REGION Network 41: Kích hoạt mô phỏng TT3208_Bon2 khi ở chế độ Sim Mode
   RUNG wire#powerrail
      Contact( "HMI_Sim_Mode" )
      Contact( "TT3208_Bon2_Sim_Req" )
      Coil( "TT3208_Bon2_Sim_Active" )
   END_RUNG
   // the same network as SCL:
   "TT3208_Bon2_Sim_Active" := "HMI_Sim_Mode" AND "TT3208_Bon2_Sim_Req";
END_REGION

REGION Network 42: Đọc giá trị mô phỏng TT3208_Bon2 vào hiệu dụng
   RUNG wire#powerrail
      Contact( "TT3208_Bon2_Sim_Active" )
      { S7_GenerateENO := "TRUE" } Move(in := "TT3208_Bon2_HMI", out1 => "TT3208_Bon2_Eff")
   END_RUNG
   // the same network as SCL:
   IF "TT3208_Bon2_Sim_Active" THEN "TT3208_Bon2_Eff" := "TT3208_Bon2_HMI"; END_IF;
END_REGION

REGION Network 43: Đọc giá trị vật lý TT3208_Bon2 vào hiệu dụng
   RUNG wire#powerrail
      I_Contact( "TT3208_Bon2_Sim_Active" )
      { S7_GenerateENO := "TRUE" } Move(in := "TT3208_Bon2", out1 => "TT3208_Bon2_Eff")
   END_RUNG
   // the same network as SCL:
   IF NOT "TT3208_Bon2_Sim_Active" THEN "TT3208_Bon2_Eff" := "TT3208_Bon2"; END_IF;
END_REGION

REGION Network 44: Kiểm tra hợp lệ Setpoint PLC1
   RUNG wire#powerrail
      { S7_Templates := "SrcType := Real" } GT_Contact(in1 := "HMI_SP_PLC1_Nuoc_Bon1", in2 := 0.0)
      { S7_Templates := "SrcType := Real" } GT_Contact(in1 := "HMI_SP_PLC1_Nuoc_Bon2", in2 := 0.0)
      { S7_Templates := "SrcType := Real" } GT_Contact(in1 := "HMI_SP_PLC1_Toc_Do_Bon1", in2 := 0.0)
      { S7_Templates := "SrcType := Real" } GT_Contact(in1 := "HMI_SP_PLC1_Toc_Do_Bon2_Main", in2 := 0.0)
      { S7_Templates := "SrcType := Real" } GT_Contact(in1 := "HMI_SP_PLC1_Nhiet_Do_Bon2", in2 := 0.0)
      { S7_Templates := "SrcType := Time" } GT_Contact(in1 := "HMI_SP_Time_Khuay_Bon1", in2 := T#0s)
      { S7_Templates := "SrcType := Time" } GT_Contact(in1 := "HMI_SP_Time_Fwd", in2 := T#0s)
      { S7_Templates := "SrcType := Time" } GT_Contact(in1 := "HMI_SP_Time_Rev", in2 := T#0s)
      { S7_Templates := "SrcType := Time" } GT_Contact(in1 := "HMI_SP_Time_Sterilize", in2 := T#0s)
      Coil( "PLC1_SP_Valid" )
   END_RUNG
   // the same network as SCL:
   "PLC1_SP_Valid" := ("HMI_SP_PLC1_Nuoc_Bon1" > 0.0) AND ("HMI_SP_PLC1_Nuoc_Bon2" > 0.0) AND ("HMI_SP_PLC1_Toc_Do_Bon1" > 0.0) AND ("HMI_SP_PLC1_Toc_Do_Bon2_Main" > 0.0) AND ("HMI_SP_PLC1_Nhiet_Do_Bon2" > 0.0) AND ("HMI_SP_Time_Khuay_Bon1" > T#0s) AND ("HMI_SP_Time_Fwd" > T#0s) AND ("HMI_SP_Time_Rev" > T#0s) AND ("HMI_SP_Time_Sterilize" > T#0s);
END_REGION

REGION Network 45: Nhận cạnh lên nút nhấn Start PLC1
   RUNG wire#powerrail
      Contact( "Nut_Khoi_Dong_Eff" )
      P_Trig( "PLC1_Start_Edge_Old" )
      Coil( "PLC1_Start_Edge_Edge" )
   END_RUNG
   // the same network as SCL:
   #_w1 := "Nut_Khoi_Dong_Eff" AND NOT "PLC1_Start_Edge_Old";   // rising edge
   "PLC1_Start_Edge_Old" := "Nut_Khoi_Dong_Eff";
   "PLC1_Start_Edge_Edge" := #_w1;
END_REGION

REGION Network 46: Khởi động chu trình PLC1 - Set Auto Enable
   RUNG wire#powerrail
      { S7_Templates := "SrcType := Int" } EQ_Contact(in1 := "PLC1_State", in2 := 0)
      Contact( "PLC1_Start_Edge_Edge" )
      I_Contact( "PLC1_Loi_Tong" )
      Contact( "PLC1_SP_Valid" )
      S_Coil( "PLC1_Auto_Enable" )
   END_RUNG
   // the same network as SCL:
   IF ("PLC1_State" = 0) AND "PLC1_Start_Edge_Edge" AND NOT "PLC1_Loi_Tong" AND "PLC1_SP_Valid" THEN
       "PLC1_Auto_Enable" := TRUE;
   END_IF;
END_REGION

REGION Network 47: Khởi động chu trình PLC1 - Chuyển sang State 10
   RUNG wire#powerrail
      { S7_Templates := "SrcType := Int" } EQ_Contact(in1 := "PLC1_State", in2 := 0)
      Contact( "PLC1_Start_Edge_Edge" )
      I_Contact( "PLC1_Loi_Tong" )
      Contact( "PLC1_SP_Valid" )
      { S7_GenerateENO := "TRUE" } Move(in := 10, out1 => "PLC1_State")
   END_RUNG
   // the same network as SCL:
   IF ("PLC1_State" = 0) AND "PLC1_Start_Edge_Edge" AND NOT "PLC1_Loi_Tong" AND "PLC1_SP_Valid" THEN
       "PLC1_State" := 10;
   END_IF;
END_REGION

REGION Network 48: Báo lỗi setpoint PLC1 khi bấm Start
   RUNG wire#powerrail
      Contact( "PLC1_Start_Edge_Edge" )
      I_Contact( "PLC1_Loi_Tong" )
      I_Contact( "PLC1_SP_Valid" )
      S_Coil( "PLC1_Loi_Setpoint" )
   END_RUNG
   // the same network as SCL:
   IF "PLC1_Start_Edge_Edge" AND NOT "PLC1_Loi_Tong" AND NOT "PLC1_SP_Valid" THEN
       "PLC1_Loi_Setpoint" := TRUE;
   END_IF;
END_REGION

REGION Network 49: Stop PLC1 từ nút vật lý hoặc HMI
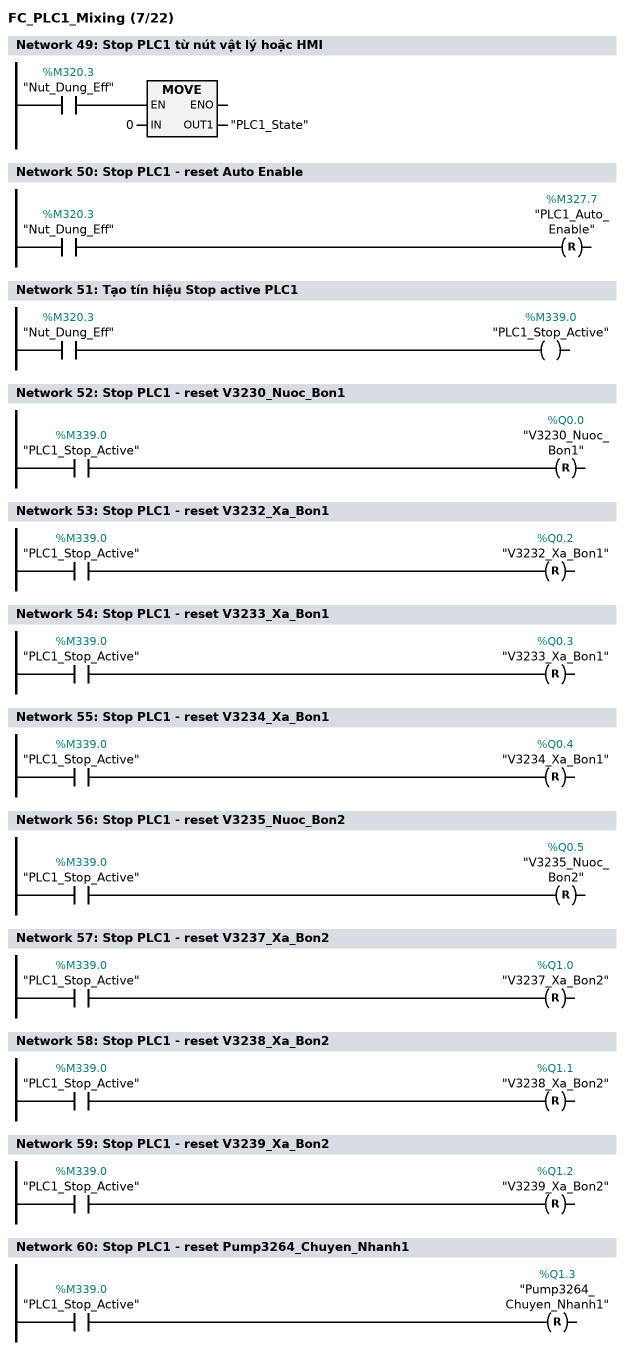
   RUNG wire#powerrail
      Contact( "Nut_Dung_Eff" )
      { S7_GenerateENO := "TRUE" } Move(in := 0, out1 => "PLC1_State")
   END_RUNG
   // the same network as SCL:
   IF "Nut_Dung_Eff" THEN "PLC1_State" := 0; END_IF;
END_REGION

REGION Network 50: Stop PLC1 - reset Auto Enable
   RUNG wire#powerrail
      Contact( "Nut_Dung_Eff" )
      R_Coil( "PLC1_Auto_Enable" )
   END_RUNG
   // the same network as SCL:
   IF "Nut_Dung_Eff" THEN "PLC1_Auto_Enable" := FALSE; END_IF;
END_REGION

REGION Network 51: Tạo tín hiệu Stop active PLC1
   RUNG wire#powerrail
      Contact( "Nut_Dung_Eff" )
      Coil( "PLC1_Stop_Active" )
   END_RUNG
   // the same network as SCL:
   "PLC1_Stop_Active" := "Nut_Dung_Eff";
END_REGION

REGION Network 52: Stop PLC1 - reset V3230_Nuoc_Bon1
   RUNG wire#powerrail
      Contact( "PLC1_Stop_Active" )
      R_Coil( "V3230_Nuoc_Bon1" )
   END_RUNG
   // the same network as SCL:
   IF "PLC1_Stop_Active" THEN "V3230_Nuoc_Bon1" := FALSE; END_IF;
END_REGION

REGION Network 53: Stop PLC1 - reset V3232_Xa_Bon1
   RUNG wire#powerrail
      Contact( "PLC1_Stop_Active" )
      R_Coil( "V3232_Xa_Bon1" )
   END_RUNG
   // the same network as SCL:
   IF "PLC1_Stop_Active" THEN "V3232_Xa_Bon1" := FALSE; END_IF;
END_REGION

REGION Network 54: Stop PLC1 - reset V3233_Xa_Bon1
   RUNG wire#powerrail
      Contact( "PLC1_Stop_Active" )
      R_Coil( "V3233_Xa_Bon1" )
   END_RUNG
   // the same network as SCL:
   IF "PLC1_Stop_Active" THEN "V3233_Xa_Bon1" := FALSE; END_IF;
END_REGION

REGION Network 55: Stop PLC1 - reset V3234_Xa_Bon1
   RUNG wire#powerrail
      Contact( "PLC1_Stop_Active" )
      R_Coil( "V3234_Xa_Bon1" )
   END_RUNG
   // the same network as SCL:
   IF "PLC1_Stop_Active" THEN "V3234_Xa_Bon1" := FALSE; END_IF;
END_REGION

REGION Network 56: Stop PLC1 - reset V3235_Nuoc_Bon2
   RUNG wire#powerrail
      Contact( "PLC1_Stop_Active" )
      R_Coil( "V3235_Nuoc_Bon2" )
   END_RUNG
   // the same network as SCL:
   IF "PLC1_Stop_Active" THEN "V3235_Nuoc_Bon2" := FALSE; END_IF;
END_REGION

REGION Network 57: Stop PLC1 - reset V3237_Xa_Bon2
   RUNG wire#powerrail
      Contact( "PLC1_Stop_Active" )
      R_Coil( "V3237_Xa_Bon2" )
   END_RUNG
   // the same network as SCL:
   IF "PLC1_Stop_Active" THEN "V3237_Xa_Bon2" := FALSE; END_IF;
END_REGION

REGION Network 58: Stop PLC1 - reset V3238_Xa_Bon2
   RUNG wire#powerrail
      Contact( "PLC1_Stop_Active" )
      R_Coil( "V3238_Xa_Bon2" )
   END_RUNG
   // the same network as SCL:
   IF "PLC1_Stop_Active" THEN "V3238_Xa_Bon2" := FALSE; END_IF;
END_REGION

REGION Network 59: Stop PLC1 - reset V3239_Xa_Bon2
   RUNG wire#powerrail
      Contact( "PLC1_Stop_Active" )
      R_Coil( "V3239_Xa_Bon2" )
   END_RUNG
   // the same network as SCL:
   IF "PLC1_Stop_Active" THEN "V3239_Xa_Bon2" := FALSE; END_IF;
END_REGION

REGION Network 60: Stop PLC1 - reset Pump3264_Chuyen_Nhanh1
   RUNG wire#powerrail
      Contact( "PLC1_Stop_Active" )
      R_Coil( "Pump3264_Chuyen_Nhanh1" )
   END_RUNG
   // the same network as SCL:
   IF "PLC1_Stop_Active" THEN "Pump3264_Chuyen_Nhanh1" := FALSE; END_IF;
END_REGION

REGION Network 61: Stop PLC1 - reset PID Enable
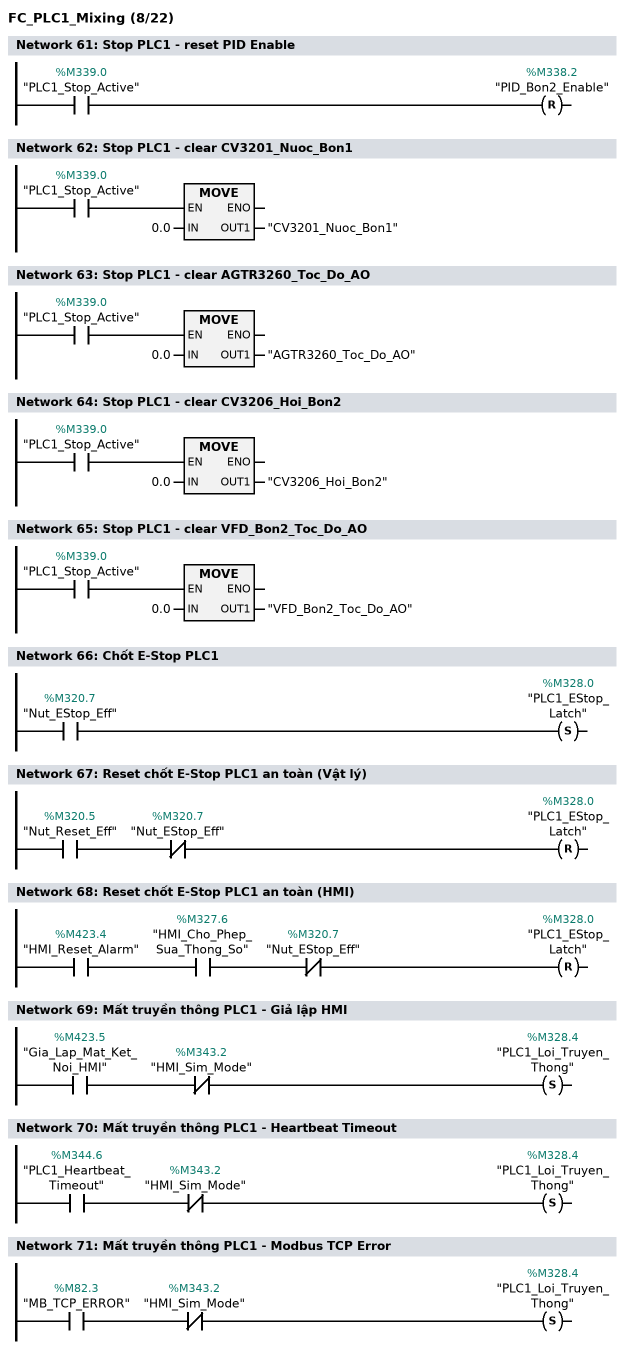
   RUNG wire#powerrail
      Contact( "PLC1_Stop_Active" )
      R_Coil( "PID_Bon2_Enable" )
   END_RUNG
   // the same network as SCL:
   IF "PLC1_Stop_Active" THEN "PID_Bon2_Enable" := FALSE; END_IF;
END_REGION

REGION Network 62: Stop PLC1 - clear CV3201_Nuoc_Bon1
   RUNG wire#powerrail
      Contact( "PLC1_Stop_Active" )
      { S7_GenerateENO := "TRUE" } Move(in := 0.0, out1 => "CV3201_Nuoc_Bon1")
   END_RUNG
   // the same network as SCL:
   IF "PLC1_Stop_Active" THEN "CV3201_Nuoc_Bon1" := 0.0; END_IF;
END_REGION

REGION Network 63: Stop PLC1 - clear AGTR3260_Toc_Do_AO
   RUNG wire#powerrail
      Contact( "PLC1_Stop_Active" )
      { S7_GenerateENO := "TRUE" } Move(in := 0.0, out1 => "AGTR3260_Toc_Do_AO")
   END_RUNG
   // the same network as SCL:
   IF "PLC1_Stop_Active" THEN "AGTR3260_Toc_Do_AO" := 0.0; END_IF;
END_REGION

REGION Network 64: Stop PLC1 - clear CV3206_Hoi_Bon2
   RUNG wire#powerrail
      Contact( "PLC1_Stop_Active" )
      { S7_GenerateENO := "TRUE" } Move(in := 0.0, out1 => "CV3206_Hoi_Bon2")
   END_RUNG
   // the same network as SCL:
   IF "PLC1_Stop_Active" THEN "CV3206_Hoi_Bon2" := 0.0; END_IF;
END_REGION

REGION Network 65: Stop PLC1 - clear VFD_Bon2_Toc_Do_AO
   RUNG wire#powerrail
      Contact( "PLC1_Stop_Active" )
      { S7_GenerateENO := "TRUE" } Move(in := 0.0, out1 => "VFD_Bon2_Toc_Do_AO")
   END_RUNG
   // the same network as SCL:
   IF "PLC1_Stop_Active" THEN "VFD_Bon2_Toc_Do_AO" := 0.0; END_IF;
END_REGION

REGION Network 66: Chốt E-Stop PLC1
   RUNG wire#powerrail
      Contact( "Nut_EStop_Eff" )
      S_Coil( "PLC1_EStop_Latch" )
   END_RUNG
   // the same network as SCL:
   IF "Nut_EStop_Eff" THEN "PLC1_EStop_Latch" := TRUE; END_IF;
END_REGION

REGION Network 67: Reset chốt E-Stop PLC1 an toàn (Vật lý)
   RUNG wire#powerrail
      Contact( "Nut_Reset_Eff" )
      I_Contact( "Nut_EStop_Eff" )
      R_Coil( "PLC1_EStop_Latch" )
   END_RUNG
   // the same network as SCL:
   IF "Nut_Reset_Eff" AND NOT "Nut_EStop_Eff" THEN "PLC1_EStop_Latch" := FALSE; END_IF;
END_REGION

REGION Network 68: Reset chốt E-Stop PLC1 an toàn (HMI)
   RUNG wire#powerrail
      Contact( "HMI_Reset_Alarm" )
      Contact( "HMI_Cho_Phep_Sua_Thong_So" )
      I_Contact( "Nut_EStop_Eff" )
      R_Coil( "PLC1_EStop_Latch" )
   END_RUNG
   // the same network as SCL:
   IF "HMI_Reset_Alarm" AND "HMI_Cho_Phep_Sua_Thong_So" AND NOT "Nut_EStop_Eff" THEN
       "PLC1_EStop_Latch" := FALSE;
   END_IF;
END_REGION

REGION Network 69: Mất truyền thông PLC1 - Giả lập HMI
   RUNG wire#powerrail
      Contact( "Gia_Lap_Mat_Ket_Noi_HMI" )
      I_Contact( "HMI_Sim_Mode" )
      S_Coil( "PLC1_Loi_Truyen_Thong" )
   END_RUNG
   // the same network as SCL:
   IF "Gia_Lap_Mat_Ket_Noi_HMI" AND NOT "HMI_Sim_Mode" THEN "PLC1_Loi_Truyen_Thong" := TRUE; END_IF;
END_REGION

REGION Network 70: Mất truyền thông PLC1 - Heartbeat Timeout
   RUNG wire#powerrail
      Contact( "PLC1_Heartbeat_Timeout" )
      I_Contact( "HMI_Sim_Mode" )
      S_Coil( "PLC1_Loi_Truyen_Thong" )
   END_RUNG
   // the same network as SCL:
   IF "PLC1_Heartbeat_Timeout" AND NOT "HMI_Sim_Mode" THEN "PLC1_Loi_Truyen_Thong" := TRUE; END_IF;
END_REGION

REGION Network 71: Mất truyền thông PLC1 - Modbus TCP Error
   RUNG wire#powerrail
      Contact( "MB_TCP_ERROR" )
      I_Contact( "HMI_Sim_Mode" )
      S_Coil( "PLC1_Loi_Truyen_Thong" )
   END_RUNG
   // the same network as SCL:
   IF "MB_TCP_ERROR" AND NOT "HMI_Sim_Mode" THEN "PLC1_Loi_Truyen_Thong" := TRUE; END_IF;
END_REGION

REGION Network 72: Dry Run bơm Nhánh 1
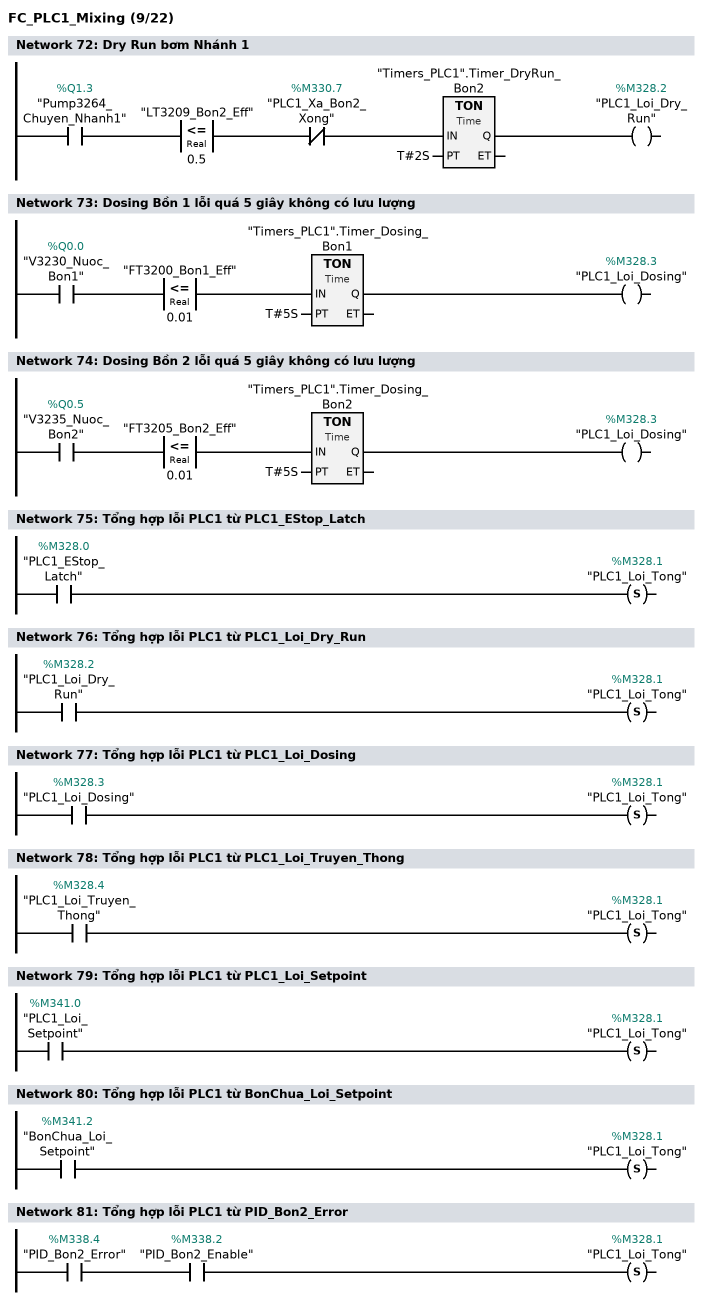
   RUNG wire#powerrail
      Contact( "Pump3264_Chuyen_Nhanh1" )
      { S7_Templates := "SrcType := Real" } LE_Contact(in1 := "LT3209_Bon2_Eff", in2 := 0.5)
      I_Contact( "PLC1_Xa_Bon2_Xong" )
      { S7_Templates := "time_type := Time" } "Timers_PLC1".Timer_DryRun_Bon2.TON(pt := T#2S, et =>)
      Coil( "PLC1_Loi_Dry_Run" )
   END_RUNG
   // the same network as SCL:
   "Timers_PLC1".Timer_DryRun_Bon2.TON(IN := "Pump3264_Chuyen_Nhanh1" AND ("LT3209_Bon2_Eff" <= 0.5) AND NOT "PLC1_Xa_Bon2_Xong",
                           PT := T#2S);
   "PLC1_Loi_Dry_Run" := "Timers_PLC1".Timer_DryRun_Bon2.Q;
END_REGION

REGION Network 73: Dosing Bồn 1 lỗi quá 5 giây không có lưu lượng
   RUNG wire#powerrail
      Contact( "V3230_Nuoc_Bon1" )
      { S7_Templates := "SrcType := Real" } LE_Contact(in1 := "FT3200_Bon1_Eff", in2 := 0.01)
      { S7_Templates := "time_type := Time" } "Timers_PLC1".Timer_Dosing_Bon1.TON(pt := T#5S, et =>)
      Coil( "PLC1_Loi_Dosing" )
   END_RUNG
   // the same network as SCL:
   "Timers_PLC1".Timer_Dosing_Bon1.TON(IN := "V3230_Nuoc_Bon1" AND ("FT3200_Bon1_Eff" <= 0.01), PT := T#5S);
   "PLC1_Loi_Dosing" := "Timers_PLC1".Timer_Dosing_Bon1.Q;
END_REGION

REGION Network 74: Dosing Bồn 2 lỗi quá 5 giây không có lưu lượng
   RUNG wire#powerrail
      Contact( "V3235_Nuoc_Bon2" )
      { S7_Templates := "SrcType := Real" } LE_Contact(in1 := "FT3205_Bon2_Eff", in2 := 0.01)
      { S7_Templates := "time_type := Time" } "Timers_PLC1".Timer_Dosing_Bon2.TON(pt := T#5S, et =>)
      Coil( "PLC1_Loi_Dosing" )
   END_RUNG
   // the same network as SCL:
   "Timers_PLC1".Timer_Dosing_Bon2.TON(IN := "V3235_Nuoc_Bon2" AND ("FT3205_Bon2_Eff" <= 0.01), PT := T#5S);
   "PLC1_Loi_Dosing" := "Timers_PLC1".Timer_Dosing_Bon2.Q;
END_REGION

REGION Network 75: Tổng hợp lỗi PLC1 từ PLC1_EStop_Latch
   RUNG wire#powerrail
      Contact( "PLC1_EStop_Latch" )
      S_Coil( "PLC1_Loi_Tong" )
   END_RUNG
   // the same network as SCL:
   IF "PLC1_EStop_Latch" THEN "PLC1_Loi_Tong" := TRUE; END_IF;
END_REGION

REGION Network 76: Tổng hợp lỗi PLC1 từ PLC1_Loi_Dry_Run
   RUNG wire#powerrail
      Contact( "PLC1_Loi_Dry_Run" )
      S_Coil( "PLC1_Loi_Tong" )
   END_RUNG
   // the same network as SCL:
   IF "PLC1_Loi_Dry_Run" THEN "PLC1_Loi_Tong" := TRUE; END_IF;
END_REGION

REGION Network 77: Tổng hợp lỗi PLC1 từ PLC1_Loi_Dosing
   RUNG wire#powerrail
      Contact( "PLC1_Loi_Dosing" )
      S_Coil( "PLC1_Loi_Tong" )
   END_RUNG
   // the same network as SCL:
   IF "PLC1_Loi_Dosing" THEN "PLC1_Loi_Tong" := TRUE; END_IF;
END_REGION

REGION Network 78: Tổng hợp lỗi PLC1 từ PLC1_Loi_Truyen_Thong
   RUNG wire#powerrail
      Contact( "PLC1_Loi_Truyen_Thong" )
      S_Coil( "PLC1_Loi_Tong" )
   END_RUNG
   // the same network as SCL:
   IF "PLC1_Loi_Truyen_Thong" THEN "PLC1_Loi_Tong" := TRUE; END_IF;
END_REGION

REGION Network 79: Tổng hợp lỗi PLC1 từ PLC1_Loi_Setpoint
   RUNG wire#powerrail
      Contact( "PLC1_Loi_Setpoint" )
      S_Coil( "PLC1_Loi_Tong" )
   END_RUNG
   // the same network as SCL:
   IF "PLC1_Loi_Setpoint" THEN "PLC1_Loi_Tong" := TRUE; END_IF;
END_REGION

REGION Network 80: Tổng hợp lỗi PLC1 từ BonChua_Loi_Setpoint
   RUNG wire#powerrail
      Contact( "BonChua_Loi_Setpoint" )
      S_Coil( "PLC1_Loi_Tong" )
   END_RUNG
   // the same network as SCL:
   IF "BonChua_Loi_Setpoint" THEN "PLC1_Loi_Tong" := TRUE; END_IF;
END_REGION

REGION Network 81: Tổng hợp lỗi PLC1 từ PID_Bon2_Error
   RUNG wire#powerrail
      Contact( "PID_Bon2_Error" )
      Contact( "PID_Bon2_Enable" )
      S_Coil( "PLC1_Loi_Tong" )
   END_RUNG
   // the same network as SCL:
   IF "PID_Bon2_Error" AND "PID_Bon2_Enable" THEN "PLC1_Loi_Tong" := TRUE; END_IF;
END_REGION

REGION Network 82: Tổng hợp lỗi PLC1 từ VFD_Bon2_MB_Error
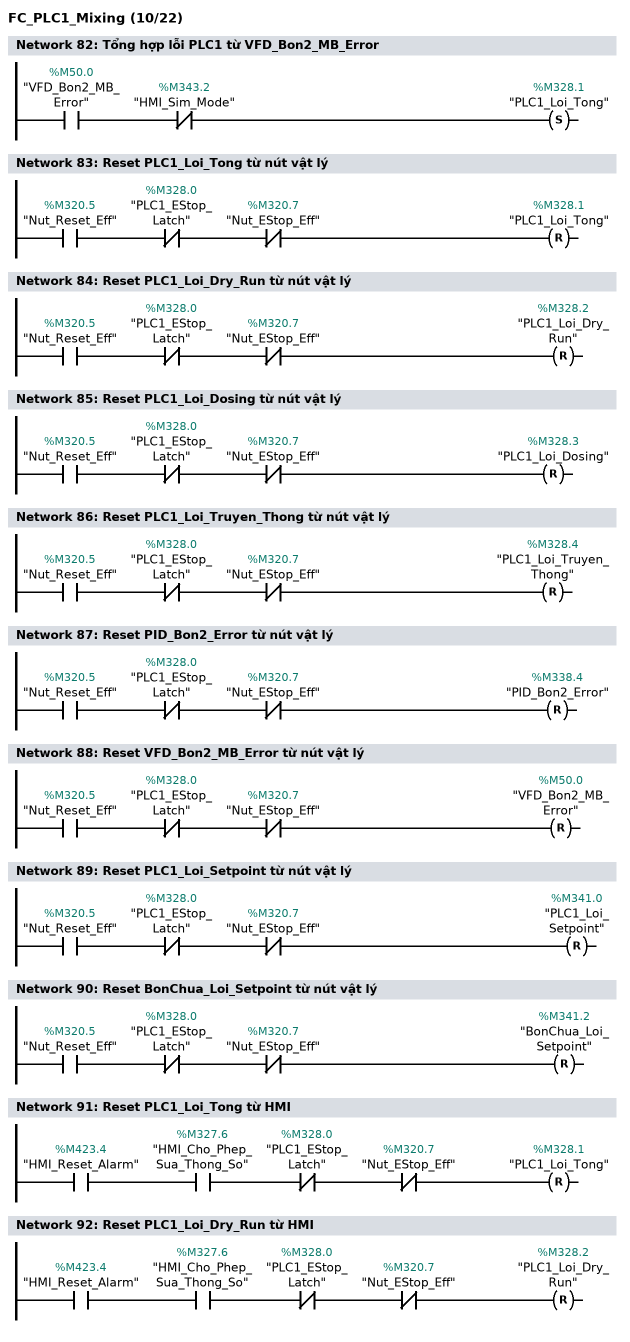
   RUNG wire#powerrail
      Contact( "VFD_Bon2_MB_Error" )
      I_Contact( "HMI_Sim_Mode" )
      S_Coil( "PLC1_Loi_Tong" )
   END_RUNG
   // the same network as SCL:
   IF "VFD_Bon2_MB_Error" AND NOT "HMI_Sim_Mode" THEN "PLC1_Loi_Tong" := TRUE; END_IF;
END_REGION

REGION Network 83: Reset PLC1_Loi_Tong từ nút vật lý
   RUNG wire#powerrail
      Contact( "Nut_Reset_Eff" )
      I_Contact( "PLC1_EStop_Latch" )
      I_Contact( "Nut_EStop_Eff" )
      R_Coil( "PLC1_Loi_Tong" )
   END_RUNG
   // the same network as SCL:
   IF "Nut_Reset_Eff" AND NOT "PLC1_EStop_Latch" AND NOT "Nut_EStop_Eff" THEN
       "PLC1_Loi_Tong" := FALSE;
   END_IF;
END_REGION

REGION Network 84: Reset PLC1_Loi_Dry_Run từ nút vật lý
   RUNG wire#powerrail
      Contact( "Nut_Reset_Eff" )
      I_Contact( "PLC1_EStop_Latch" )
      I_Contact( "Nut_EStop_Eff" )
      R_Coil( "PLC1_Loi_Dry_Run" )
   END_RUNG
   // the same network as SCL:
   IF "Nut_Reset_Eff" AND NOT "PLC1_EStop_Latch" AND NOT "Nut_EStop_Eff" THEN
       "PLC1_Loi_Dry_Run" := FALSE;
   END_IF;
END_REGION

REGION Network 85: Reset PLC1_Loi_Dosing từ nút vật lý
   RUNG wire#powerrail
      Contact( "Nut_Reset_Eff" )
      I_Contact( "PLC1_EStop_Latch" )
      I_Contact( "Nut_EStop_Eff" )
      R_Coil( "PLC1_Loi_Dosing" )
   END_RUNG
   // the same network as SCL:
   IF "Nut_Reset_Eff" AND NOT "PLC1_EStop_Latch" AND NOT "Nut_EStop_Eff" THEN
       "PLC1_Loi_Dosing" := FALSE;
   END_IF;
END_REGION

REGION Network 86: Reset PLC1_Loi_Truyen_Thong từ nút vật lý
   RUNG wire#powerrail
      Contact( "Nut_Reset_Eff" )
      I_Contact( "PLC1_EStop_Latch" )
      I_Contact( "Nut_EStop_Eff" )
      R_Coil( "PLC1_Loi_Truyen_Thong" )
   END_RUNG
   // the same network as SCL:
   IF "Nut_Reset_Eff" AND NOT "PLC1_EStop_Latch" AND NOT "Nut_EStop_Eff" THEN
       "PLC1_Loi_Truyen_Thong" := FALSE;
   END_IF;
END_REGION

REGION Network 87: Reset PID_Bon2_Error từ nút vật lý
   RUNG wire#powerrail
      Contact( "Nut_Reset_Eff" )
      I_Contact( "PLC1_EStop_Latch" )
      I_Contact( "Nut_EStop_Eff" )
      R_Coil( "PID_Bon2_Error" )
   END_RUNG
   // the same network as SCL:
   IF "Nut_Reset_Eff" AND NOT "PLC1_EStop_Latch" AND NOT "Nut_EStop_Eff" THEN
       "PID_Bon2_Error" := FALSE;
   END_IF;
END_REGION

REGION Network 88: Reset VFD_Bon2_MB_Error từ nút vật lý
   RUNG wire#powerrail
      Contact( "Nut_Reset_Eff" )
      I_Contact( "PLC1_EStop_Latch" )
      I_Contact( "Nut_EStop_Eff" )
      R_Coil( "VFD_Bon2_MB_Error" )
   END_RUNG
   // the same network as SCL:
   IF "Nut_Reset_Eff" AND NOT "PLC1_EStop_Latch" AND NOT "Nut_EStop_Eff" THEN
       "VFD_Bon2_MB_Error" := FALSE;
   END_IF;
END_REGION

REGION Network 89: Reset PLC1_Loi_Setpoint từ nút vật lý
   RUNG wire#powerrail
      Contact( "Nut_Reset_Eff" )
      I_Contact( "PLC1_EStop_Latch" )
      I_Contact( "Nut_EStop_Eff" )
      R_Coil( "PLC1_Loi_Setpoint" )
   END_RUNG
   // the same network as SCL:
   IF "Nut_Reset_Eff" AND NOT "PLC1_EStop_Latch" AND NOT "Nut_EStop_Eff" THEN
       "PLC1_Loi_Setpoint" := FALSE;
   END_IF;
END_REGION

REGION Network 90: Reset BonChua_Loi_Setpoint từ nút vật lý
   RUNG wire#powerrail
      Contact( "Nut_Reset_Eff" )
      I_Contact( "PLC1_EStop_Latch" )
      I_Contact( "Nut_EStop_Eff" )
      R_Coil( "BonChua_Loi_Setpoint" )
   END_RUNG
   // the same network as SCL:
   IF "Nut_Reset_Eff" AND NOT "PLC1_EStop_Latch" AND NOT "Nut_EStop_Eff" THEN
       "BonChua_Loi_Setpoint" := FALSE;
   END_IF;
END_REGION

REGION Network 91: Reset PLC1_Loi_Tong từ HMI
   RUNG wire#powerrail
      Contact( "HMI_Reset_Alarm" )
      Contact( "HMI_Cho_Phep_Sua_Thong_So" )
      I_Contact( "PLC1_EStop_Latch" )
      I_Contact( "Nut_EStop_Eff" )
      R_Coil( "PLC1_Loi_Tong" )
   END_RUNG
   // the same network as SCL:
   IF "HMI_Reset_Alarm" AND "HMI_Cho_Phep_Sua_Thong_So" AND NOT "PLC1_EStop_Latch" AND NOT "Nut_EStop_Eff" THEN
       "PLC1_Loi_Tong" := FALSE;
   END_IF;
END_REGION

REGION Network 92: Reset PLC1_Loi_Dry_Run từ HMI
   RUNG wire#powerrail
      Contact( "HMI_Reset_Alarm" )
      Contact( "HMI_Cho_Phep_Sua_Thong_So" )
      I_Contact( "PLC1_EStop_Latch" )
      I_Contact( "Nut_EStop_Eff" )
      R_Coil( "PLC1_Loi_Dry_Run" )
   END_RUNG
   // the same network as SCL:
   IF "HMI_Reset_Alarm" AND "HMI_Cho_Phep_Sua_Thong_So" AND NOT "PLC1_EStop_Latch" AND NOT "Nut_EStop_Eff" THEN
       "PLC1_Loi_Dry_Run" := FALSE;
   END_IF;
END_REGION

REGION Network 93: Reset PLC1_Loi_Dosing từ HMI
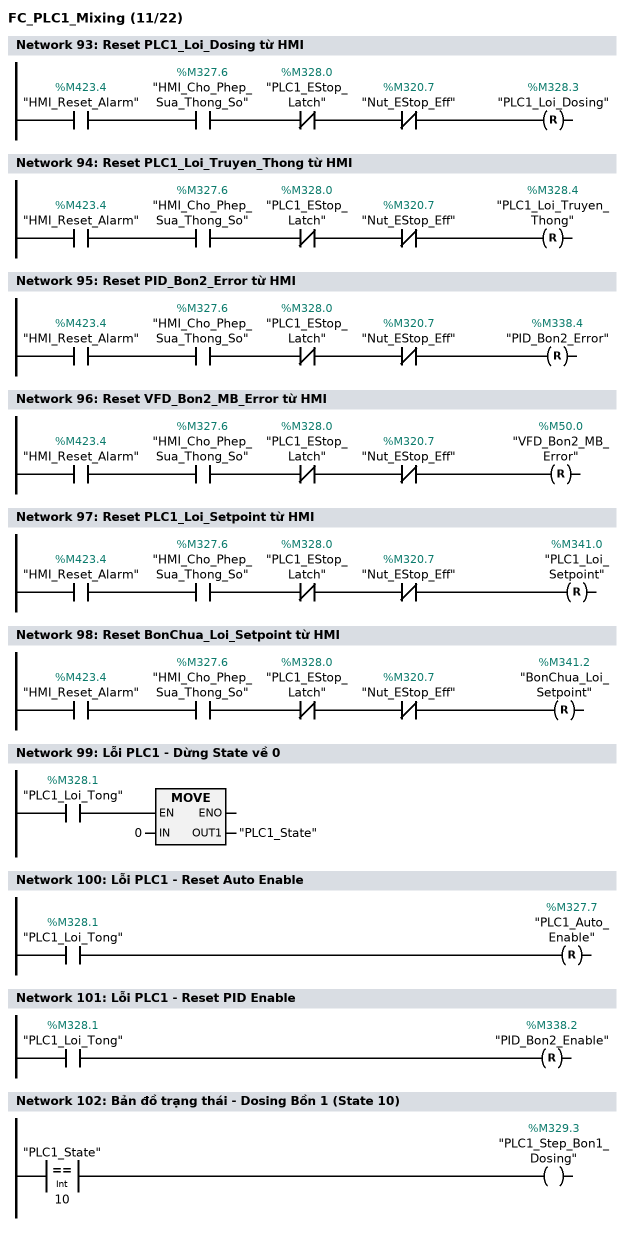
   RUNG wire#powerrail
      Contact( "HMI_Reset_Alarm" )
      Contact( "HMI_Cho_Phep_Sua_Thong_So" )
      I_Contact( "PLC1_EStop_Latch" )
      I_Contact( "Nut_EStop_Eff" )
      R_Coil( "PLC1_Loi_Dosing" )
   END_RUNG
   // the same network as SCL:
   IF "HMI_Reset_Alarm" AND "HMI_Cho_Phep_Sua_Thong_So" AND NOT "PLC1_EStop_Latch" AND NOT "Nut_EStop_Eff" THEN
       "PLC1_Loi_Dosing" := FALSE;
   END_IF;
END_REGION

REGION Network 94: Reset PLC1_Loi_Truyen_Thong từ HMI
   RUNG wire#powerrail
      Contact( "HMI_Reset_Alarm" )
      Contact( "HMI_Cho_Phep_Sua_Thong_So" )
      I_Contact( "PLC1_EStop_Latch" )
      I_Contact( "Nut_EStop_Eff" )
      R_Coil( "PLC1_Loi_Truyen_Thong" )
   END_RUNG
   // the same network as SCL:
   IF "HMI_Reset_Alarm" AND "HMI_Cho_Phep_Sua_Thong_So" AND NOT "PLC1_EStop_Latch" AND NOT "Nut_EStop_Eff" THEN
       "PLC1_Loi_Truyen_Thong" := FALSE;
   END_IF;
END_REGION

REGION Network 95: Reset PID_Bon2_Error từ HMI
   RUNG wire#powerrail
      Contact( "HMI_Reset_Alarm" )
      Contact( "HMI_Cho_Phep_Sua_Thong_So" )
      I_Contact( "PLC1_EStop_Latch" )
      I_Contact( "Nut_EStop_Eff" )
      R_Coil( "PID_Bon2_Error" )
   END_RUNG
   // the same network as SCL:
   IF "HMI_Reset_Alarm" AND "HMI_Cho_Phep_Sua_Thong_So" AND NOT "PLC1_EStop_Latch" AND NOT "Nut_EStop_Eff" THEN
       "PID_Bon2_Error" := FALSE;
   END_IF;
END_REGION

REGION Network 96: Reset VFD_Bon2_MB_Error từ HMI
   RUNG wire#powerrail
      Contact( "HMI_Reset_Alarm" )
      Contact( "HMI_Cho_Phep_Sua_Thong_So" )
      I_Contact( "PLC1_EStop_Latch" )
      I_Contact( "Nut_EStop_Eff" )
      R_Coil( "VFD_Bon2_MB_Error" )
   END_RUNG
   // the same network as SCL:
   IF "HMI_Reset_Alarm" AND "HMI_Cho_Phep_Sua_Thong_So" AND NOT "PLC1_EStop_Latch" AND NOT "Nut_EStop_Eff" THEN
       "VFD_Bon2_MB_Error" := FALSE;
   END_IF;
END_REGION

REGION Network 97: Reset PLC1_Loi_Setpoint từ HMI
   RUNG wire#powerrail
      Contact( "HMI_Reset_Alarm" )
      Contact( "HMI_Cho_Phep_Sua_Thong_So" )
      I_Contact( "PLC1_EStop_Latch" )
      I_Contact( "Nut_EStop_Eff" )
      R_Coil( "PLC1_Loi_Setpoint" )
   END_RUNG
   // the same network as SCL:
   IF "HMI_Reset_Alarm" AND "HMI_Cho_Phep_Sua_Thong_So" AND NOT "PLC1_EStop_Latch" AND NOT "Nut_EStop_Eff" THEN
       "PLC1_Loi_Setpoint" := FALSE;
   END_IF;
END_REGION

REGION Network 98: Reset BonChua_Loi_Setpoint từ HMI
   RUNG wire#powerrail
      Contact( "HMI_Reset_Alarm" )
      Contact( "HMI_Cho_Phep_Sua_Thong_So" )
      I_Contact( "PLC1_EStop_Latch" )
      I_Contact( "Nut_EStop_Eff" )
      R_Coil( "BonChua_Loi_Setpoint" )
   END_RUNG
   // the same network as SCL:
   IF "HMI_Reset_Alarm" AND "HMI_Cho_Phep_Sua_Thong_So" AND NOT "PLC1_EStop_Latch" AND NOT "Nut_EStop_Eff" THEN
       "BonChua_Loi_Setpoint" := FALSE;
   END_IF;
END_REGION

REGION Network 99: Lỗi PLC1 - Dừng State về 0
   RUNG wire#powerrail
      Contact( "PLC1_Loi_Tong" )
      { S7_GenerateENO := "TRUE" } Move(in := 0, out1 => "PLC1_State")
   END_RUNG
   // the same network as SCL:
   IF "PLC1_Loi_Tong" THEN "PLC1_State" := 0; END_IF;
END_REGION

REGION Network 100: Lỗi PLC1 - Reset Auto Enable
   RUNG wire#powerrail
      Contact( "PLC1_Loi_Tong" )
      R_Coil( "PLC1_Auto_Enable" )
   END_RUNG
   // the same network as SCL:
   IF "PLC1_Loi_Tong" THEN "PLC1_Auto_Enable" := FALSE; END_IF;
END_REGION

REGION Network 101: Lỗi PLC1 - Reset PID Enable
   RUNG wire#powerrail
      Contact( "PLC1_Loi_Tong" )
      R_Coil( "PID_Bon2_Enable" )
   END_RUNG
   // the same network as SCL:
   IF "PLC1_Loi_Tong" THEN "PID_Bon2_Enable" := FALSE; END_IF;
END_REGION

REGION Network 102: Bản đồ trạng thái - Dosing Bồn 1 (State 10)
   RUNG wire#powerrail
      { S7_Templates := "SrcType := Int" } EQ_Contact(in1 := "PLC1_State", in2 := 10)
      Coil( "PLC1_Step_Bon1_Dosing" )
   END_RUNG
   // the same network as SCL:
   "PLC1_Step_Bon1_Dosing" := "PLC1_State" = 10;
END_REGION

REGION Network 103: Bản đồ trạng thái - Tip Bồn 1 (State 11)
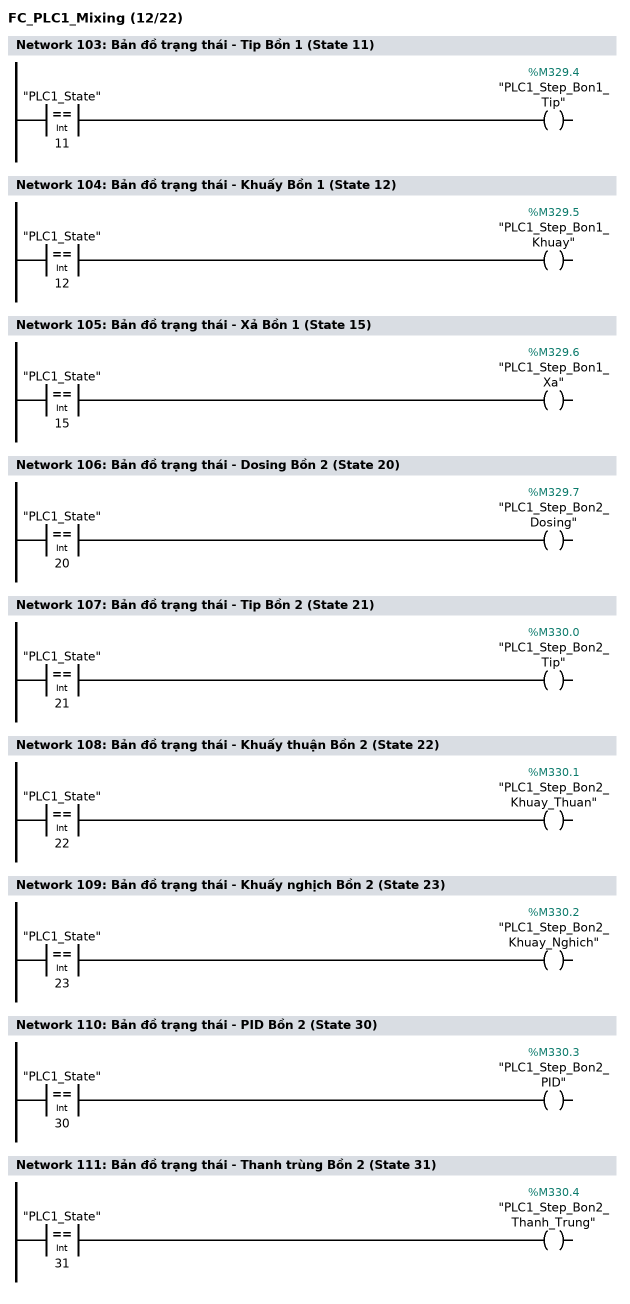
   RUNG wire#powerrail
      { S7_Templates := "SrcType := Int" } EQ_Contact(in1 := "PLC1_State", in2 := 11)
      Coil( "PLC1_Step_Bon1_Tip" )
   END_RUNG
   // the same network as SCL:
   "PLC1_Step_Bon1_Tip" := "PLC1_State" = 11;
END_REGION

REGION Network 104: Bản đồ trạng thái - Khuấy Bồn 1 (State 12)
   RUNG wire#powerrail
      { S7_Templates := "SrcType := Int" } EQ_Contact(in1 := "PLC1_State", in2 := 12)
      Coil( "PLC1_Step_Bon1_Khuay" )
   END_RUNG
   // the same network as SCL:
   "PLC1_Step_Bon1_Khuay" := "PLC1_State" = 12;
END_REGION

REGION Network 105: Bản đồ trạng thái - Xả Bồn 1 (State 15)
   RUNG wire#powerrail
      { S7_Templates := "SrcType := Int" } EQ_Contact(in1 := "PLC1_State", in2 := 15)
      Coil( "PLC1_Step_Bon1_Xa" )
   END_RUNG
   // the same network as SCL:
   "PLC1_Step_Bon1_Xa" := "PLC1_State" = 15;
END_REGION

REGION Network 106: Bản đồ trạng thái - Dosing Bồn 2 (State 20)
   RUNG wire#powerrail
      { S7_Templates := "SrcType := Int" } EQ_Contact(in1 := "PLC1_State", in2 := 20)
      Coil( "PLC1_Step_Bon2_Dosing" )
   END_RUNG
   // the same network as SCL:
   "PLC1_Step_Bon2_Dosing" := "PLC1_State" = 20;
END_REGION

REGION Network 107: Bản đồ trạng thái - Tip Bồn 2 (State 21)
   RUNG wire#powerrail
      { S7_Templates := "SrcType := Int" } EQ_Contact(in1 := "PLC1_State", in2 := 21)
      Coil( "PLC1_Step_Bon2_Tip" )
   END_RUNG
   // the same network as SCL:
   "PLC1_Step_Bon2_Tip" := "PLC1_State" = 21;
END_REGION

REGION Network 108: Bản đồ trạng thái - Khuấy thuận Bồn 2 (State 22)
   RUNG wire#powerrail
      { S7_Templates := "SrcType := Int" } EQ_Contact(in1 := "PLC1_State", in2 := 22)
      Coil( "PLC1_Step_Bon2_Khuay_Thuan" )
   END_RUNG
   // the same network as SCL:
   "PLC1_Step_Bon2_Khuay_Thuan" := "PLC1_State" = 22;
END_REGION

REGION Network 109: Bản đồ trạng thái - Khuấy nghịch Bồn 2 (State 23)
   RUNG wire#powerrail
      { S7_Templates := "SrcType := Int" } EQ_Contact(in1 := "PLC1_State", in2 := 23)
      Coil( "PLC1_Step_Bon2_Khuay_Nghich" )
   END_RUNG
   // the same network as SCL:
   "PLC1_Step_Bon2_Khuay_Nghich" := "PLC1_State" = 23;
END_REGION

REGION Network 110: Bản đồ trạng thái - PID Bồn 2 (State 30)
   RUNG wire#powerrail
      { S7_Templates := "SrcType := Int" } EQ_Contact(in1 := "PLC1_State", in2 := 30)
      Coil( "PLC1_Step_Bon2_PID" )
   END_RUNG
   // the same network as SCL:
   "PLC1_Step_Bon2_PID" := "PLC1_State" = 30;
END_REGION

REGION Network 111: Bản đồ trạng thái - Thanh trùng Bồn 2 (State 31)
   RUNG wire#powerrail
      { S7_Templates := "SrcType := Int" } EQ_Contact(in1 := "PLC1_State", in2 := 31)
      Coil( "PLC1_Step_Bon2_Thanh_Trung" )
   END_RUNG
   // the same network as SCL:
   "PLC1_Step_Bon2_Thanh_Trung" := "PLC1_State" = 31;
END_REGION

REGION Network 112: Bản đồ trạng thái - Nhánh 1 Hoàn thành (State 40)
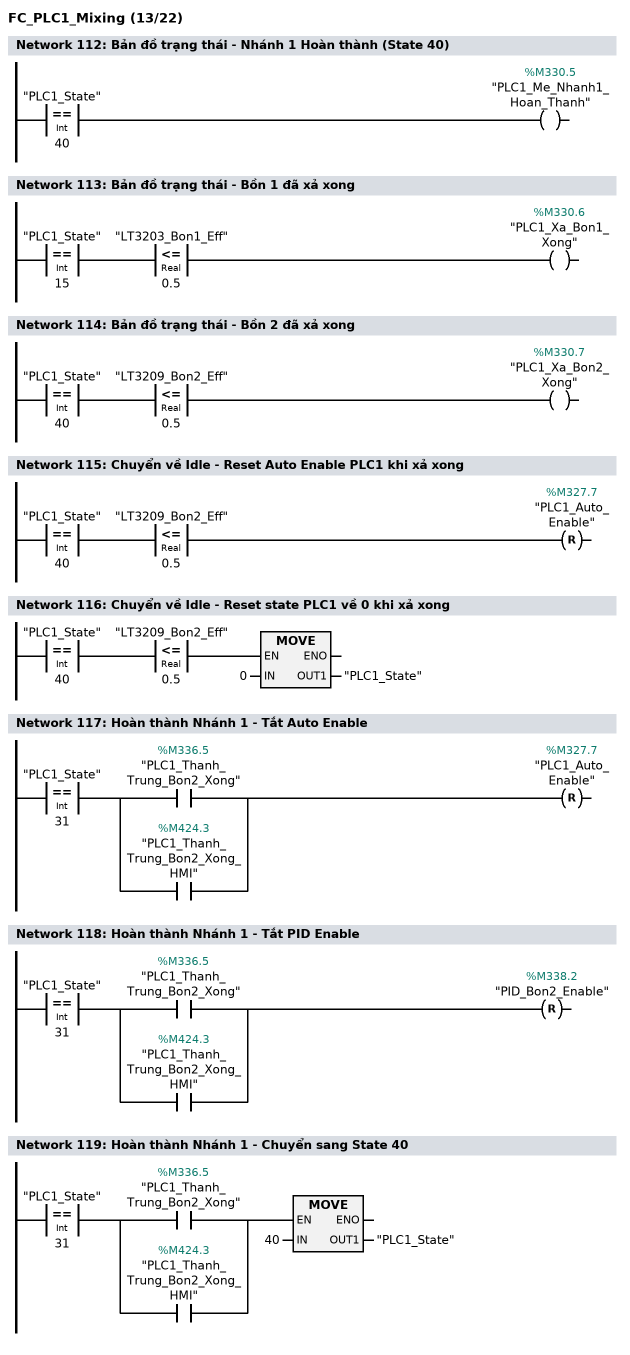
   RUNG wire#powerrail
      { S7_Templates := "SrcType := Int" } EQ_Contact(in1 := "PLC1_State", in2 := 40)
      Coil( "PLC1_Me_Nhanh1_Hoan_Thanh" )
   END_RUNG
   // the same network as SCL:
   "PLC1_Me_Nhanh1_Hoan_Thanh" := "PLC1_State" = 40;
END_REGION

REGION Network 113: Bản đồ trạng thái - Bồn 1 đã xả xong
   RUNG wire#powerrail
      { S7_Templates := "SrcType := Int" } EQ_Contact(in1 := "PLC1_State", in2 := 15)
      { S7_Templates := "SrcType := Real" } LE_Contact(in1 := "LT3203_Bon1_Eff", in2 := 0.5)
      Coil( "PLC1_Xa_Bon1_Xong" )
   END_RUNG
   // the same network as SCL:
   "PLC1_Xa_Bon1_Xong" := ("PLC1_State" = 15) AND ("LT3203_Bon1_Eff" <= 0.5);
END_REGION

REGION Network 114: Bản đồ trạng thái - Bồn 2 đã xả xong
   RUNG wire#powerrail
      { S7_Templates := "SrcType := Int" } EQ_Contact(in1 := "PLC1_State", in2 := 40)
      { S7_Templates := "SrcType := Real" } LE_Contact(in1 := "LT3209_Bon2_Eff", in2 := 0.5)
      Coil( "PLC1_Xa_Bon2_Xong" )
   END_RUNG
   // the same network as SCL:
   "PLC1_Xa_Bon2_Xong" := ("PLC1_State" = 40) AND ("LT3209_Bon2_Eff" <= 0.5);
END_REGION

REGION Network 115: Chuyển về Idle - Reset Auto Enable PLC1 khi xả xong
   RUNG wire#powerrail
      { S7_Templates := "SrcType := Int" } EQ_Contact(in1 := "PLC1_State", in2 := 40)
      { S7_Templates := "SrcType := Real" } LE_Contact(in1 := "LT3209_Bon2_Eff", in2 := 0.5)
      R_Coil( "PLC1_Auto_Enable" )
   END_RUNG
   // the same network as SCL:
   IF ("PLC1_State" = 40) AND ("LT3209_Bon2_Eff" <= 0.5) THEN "PLC1_Auto_Enable" := FALSE; END_IF;
END_REGION

REGION Network 116: Chuyển về Idle - Reset state PLC1 về 0 khi xả xong
   RUNG wire#powerrail
      { S7_Templates := "SrcType := Int" } EQ_Contact(in1 := "PLC1_State", in2 := 40)
      { S7_Templates := "SrcType := Real" } LE_Contact(in1 := "LT3209_Bon2_Eff", in2 := 0.5)
      { S7_GenerateENO := "TRUE" } Move(in := 0, out1 => "PLC1_State")
   END_RUNG
   // the same network as SCL:
   IF ("PLC1_State" = 40) AND ("LT3209_Bon2_Eff" <= 0.5) THEN "PLC1_State" := 0; END_IF;
END_REGION

REGION Network 117: Hoàn thành Nhánh 1 - Tắt Auto Enable
   RUNG wire#powerrail
      { S7_Templates := "SrcType := Int" } EQ_Contact(in1 := "PLC1_State", in2 := 31)
      wire#w1
      Contact( "PLC1_Thanh_Trung_Bon2_Xong" )
      wire#w2
      R_Coil( "PLC1_Auto_Enable" )
   END_RUNG
   RUNG wire#w1
      Contact( "PLC1_Thanh_Trung_Bon2_Xong_HMI" )
   END_RUNG wire#w2
   // the same network as SCL:
   IF ("PLC1_State" = 31) AND ("PLC1_Thanh_Trung_Bon2_Xong" OR "PLC1_Thanh_Trung_Bon2_Xong_HMI") THEN
       "PLC1_Auto_Enable" := FALSE;
   END_IF;
END_REGION

REGION Network 118: Hoàn thành Nhánh 1 - Tắt PID Enable
   RUNG wire#powerrail
      { S7_Templates := "SrcType := Int" } EQ_Contact(in1 := "PLC1_State", in2 := 31)
      wire#w1
      Contact( "PLC1_Thanh_Trung_Bon2_Xong" )
      wire#w2
      R_Coil( "PID_Bon2_Enable" )
   END_RUNG
   RUNG wire#w1
      Contact( "PLC1_Thanh_Trung_Bon2_Xong_HMI" )
   END_RUNG wire#w2
   // the same network as SCL:
   IF ("PLC1_State" = 31) AND ("PLC1_Thanh_Trung_Bon2_Xong" OR "PLC1_Thanh_Trung_Bon2_Xong_HMI") THEN
       "PID_Bon2_Enable" := FALSE;
   END_IF;
END_REGION

REGION Network 119: Hoàn thành Nhánh 1 - Chuyển sang State 40
   RUNG wire#powerrail
      { S7_Templates := "SrcType := Int" } EQ_Contact(in1 := "PLC1_State", in2 := 31)
      wire#w1
      Contact( "PLC1_Thanh_Trung_Bon2_Xong" )
      wire#w2
      { S7_GenerateENO := "TRUE" } Move(in := 40, out1 => "PLC1_State")
   END_RUNG
   RUNG wire#w1
      Contact( "PLC1_Thanh_Trung_Bon2_Xong_HMI" )
   END_RUNG wire#w2
   // the same network as SCL:
   IF ("PLC1_State" = 31) AND ("PLC1_Thanh_Trung_Bon2_Xong" OR "PLC1_Thanh_Trung_Bon2_Xong_HMI") THEN
       "PLC1_State" := 40;
   END_IF;
END_REGION

REGION Network 120: Gia nhiệt Bồn 2 đạt SP - Chuyển sang State 31
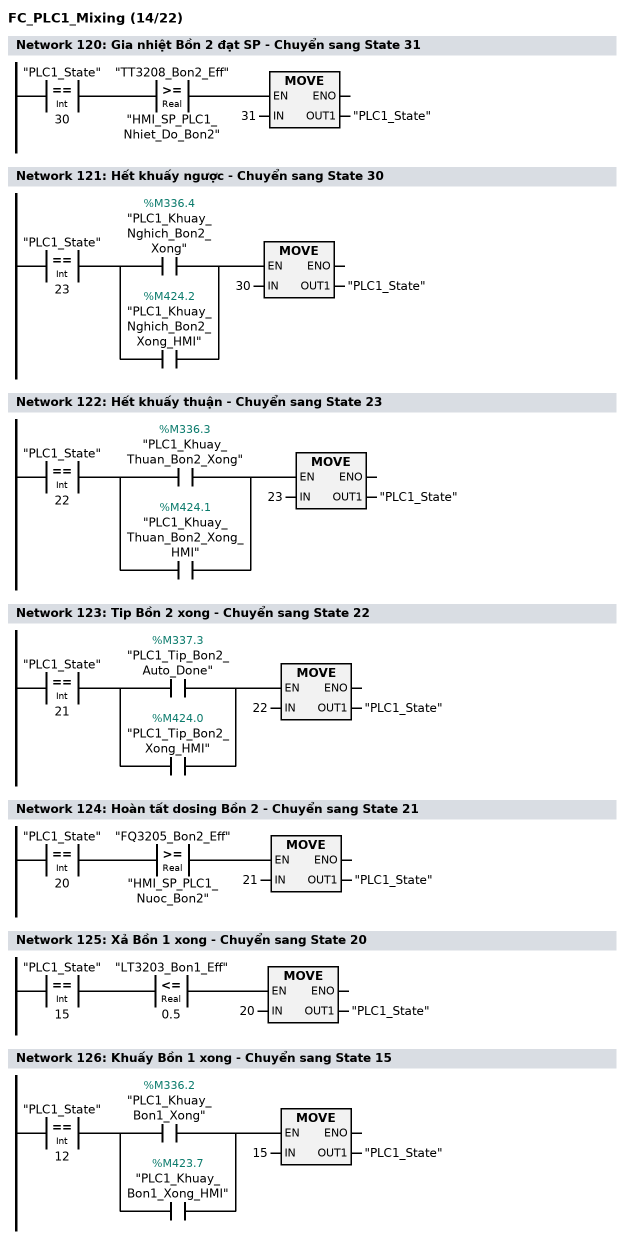
   RUNG wire#powerrail
      { S7_Templates := "SrcType := Int" } EQ_Contact(in1 := "PLC1_State", in2 := 30)
      { S7_Templates := "SrcType := Real" } GE_Contact(in1 := "TT3208_Bon2_Eff", in2 := "HMI_SP_PLC1_Nhiet_Do_Bon2")
      { S7_GenerateENO := "TRUE" } Move(in := 31, out1 => "PLC1_State")
   END_RUNG
   // the same network as SCL:
   IF ("PLC1_State" = 30) AND ("TT3208_Bon2_Eff" >= "HMI_SP_PLC1_Nhiet_Do_Bon2") THEN
       "PLC1_State" := 31;
   END_IF;
END_REGION

REGION Network 121: Hết khuấy ngược - Chuyển sang State 30
   RUNG wire#powerrail
      { S7_Templates := "SrcType := Int" } EQ_Contact(in1 := "PLC1_State", in2 := 23)
      wire#w1
      Contact( "PLC1_Khuay_Nghich_Bon2_Xong" )
      wire#w2
      { S7_GenerateENO := "TRUE" } Move(in := 30, out1 => "PLC1_State")
   END_RUNG
   RUNG wire#w1
      Contact( "PLC1_Khuay_Nghich_Bon2_Xong_HMI" )
   END_RUNG wire#w2
   // the same network as SCL:
   IF ("PLC1_State" = 23) AND ("PLC1_Khuay_Nghich_Bon2_Xong" OR "PLC1_Khuay_Nghich_Bon2_Xong_HMI") THEN
       "PLC1_State" := 30;
   END_IF;
END_REGION

REGION Network 122: Hết khuấy thuận - Chuyển sang State 23
   RUNG wire#powerrail
      { S7_Templates := "SrcType := Int" } EQ_Contact(in1 := "PLC1_State", in2 := 22)
      wire#w1
      Contact( "PLC1_Khuay_Thuan_Bon2_Xong" )
      wire#w2
      { S7_GenerateENO := "TRUE" } Move(in := 23, out1 => "PLC1_State")
   END_RUNG
   RUNG wire#w1
      Contact( "PLC1_Khuay_Thuan_Bon2_Xong_HMI" )
   END_RUNG wire#w2
   // the same network as SCL:
   IF ("PLC1_State" = 22) AND ("PLC1_Khuay_Thuan_Bon2_Xong" OR "PLC1_Khuay_Thuan_Bon2_Xong_HMI") THEN
       "PLC1_State" := 23;
   END_IF;
END_REGION

REGION Network 123: Tip Bồn 2 xong - Chuyển sang State 22
   RUNG wire#powerrail
      { S7_Templates := "SrcType := Int" } EQ_Contact(in1 := "PLC1_State", in2 := 21)
      wire#w1
      Contact( "PLC1_Tip_Bon2_Auto_Done" )
      wire#w2
      { S7_GenerateENO := "TRUE" } Move(in := 22, out1 => "PLC1_State")
   END_RUNG
   RUNG wire#w1
      Contact( "PLC1_Tip_Bon2_Xong_HMI" )
   END_RUNG wire#w2
   // the same network as SCL:
   IF ("PLC1_State" = 21) AND ("PLC1_Tip_Bon2_Auto_Done" OR "PLC1_Tip_Bon2_Xong_HMI") THEN
       "PLC1_State" := 22;
   END_IF;
END_REGION

REGION Network 124: Hoàn tất dosing Bồn 2 - Chuyển sang State 21
   RUNG wire#powerrail
      { S7_Templates := "SrcType := Int" } EQ_Contact(in1 := "PLC1_State", in2 := 20)
      { S7_Templates := "SrcType := Real" } GE_Contact(in1 := "FQ3205_Bon2_Eff", in2 := "HMI_SP_PLC1_Nuoc_Bon2")
      { S7_GenerateENO := "TRUE" } Move(in := 21, out1 => "PLC1_State")
   END_RUNG
   // the same network as SCL:
   IF ("PLC1_State" = 20) AND ("FQ3205_Bon2_Eff" >= "HMI_SP_PLC1_Nuoc_Bon2") THEN "PLC1_State" := 21; END_IF;
END_REGION

REGION Network 125: Xả Bồn 1 xong - Chuyển sang State 20
   RUNG wire#powerrail
      { S7_Templates := "SrcType := Int" } EQ_Contact(in1 := "PLC1_State", in2 := 15)
      { S7_Templates := "SrcType := Real" } LE_Contact(in1 := "LT3203_Bon1_Eff", in2 := 0.5)
      { S7_GenerateENO := "TRUE" } Move(in := 20, out1 => "PLC1_State")
   END_RUNG
   // the same network as SCL:
   IF ("PLC1_State" = 15) AND ("LT3203_Bon1_Eff" <= 0.5) THEN "PLC1_State" := 20; END_IF;
END_REGION

REGION Network 126: Khuấy Bồn 1 xong - Chuyển sang State 15
   RUNG wire#powerrail
      { S7_Templates := "SrcType := Int" } EQ_Contact(in1 := "PLC1_State", in2 := 12)
      wire#w1
      Contact( "PLC1_Khuay_Bon1_Xong" )
      wire#w2
      { S7_GenerateENO := "TRUE" } Move(in := 15, out1 => "PLC1_State")
   END_RUNG
   RUNG wire#w1
      Contact( "PLC1_Khuay_Bon1_Xong_HMI" )
   END_RUNG wire#w2
   // the same network as SCL:
   IF ("PLC1_State" = 12) AND ("PLC1_Khuay_Bon1_Xong" OR "PLC1_Khuay_Bon1_Xong_HMI") THEN
       "PLC1_State" := 15;
   END_IF;
END_REGION

REGION Network 127: Tip Bồn 1 xong - Chuyển sang State 12
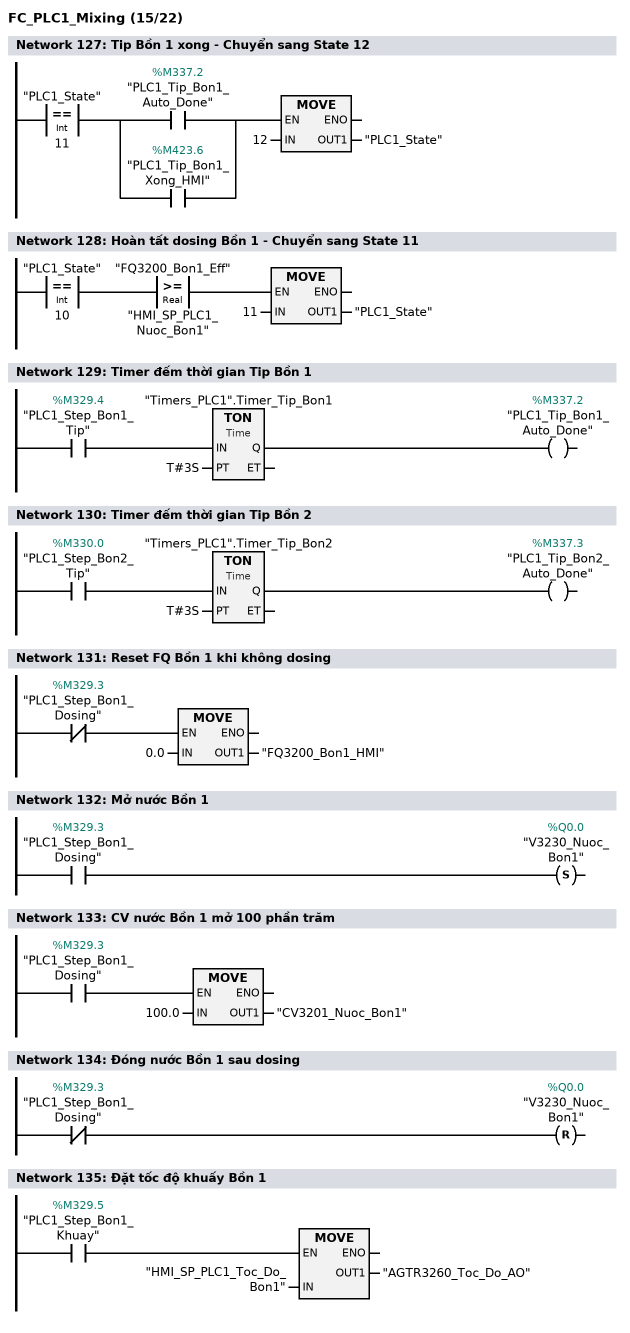
   RUNG wire#powerrail
      { S7_Templates := "SrcType := Int" } EQ_Contact(in1 := "PLC1_State", in2 := 11)
      wire#w1
      Contact( "PLC1_Tip_Bon1_Auto_Done" )
      wire#w2
      { S7_GenerateENO := "TRUE" } Move(in := 12, out1 => "PLC1_State")
   END_RUNG
   RUNG wire#w1
      Contact( "PLC1_Tip_Bon1_Xong_HMI" )
   END_RUNG wire#w2
   // the same network as SCL:
   IF ("PLC1_State" = 11) AND ("PLC1_Tip_Bon1_Auto_Done" OR "PLC1_Tip_Bon1_Xong_HMI") THEN
       "PLC1_State" := 12;
   END_IF;
END_REGION

REGION Network 128: Hoàn tất dosing Bồn 1 - Chuyển sang State 11
   RUNG wire#powerrail
      { S7_Templates := "SrcType := Int" } EQ_Contact(in1 := "PLC1_State", in2 := 10)
      { S7_Templates := "SrcType := Real" } GE_Contact(in1 := "FQ3200_Bon1_Eff", in2 := "HMI_SP_PLC1_Nuoc_Bon1")
      { S7_GenerateENO := "TRUE" } Move(in := 11, out1 => "PLC1_State")
   END_RUNG
   // the same network as SCL:
   IF ("PLC1_State" = 10) AND ("FQ3200_Bon1_Eff" >= "HMI_SP_PLC1_Nuoc_Bon1") THEN "PLC1_State" := 11; END_IF;
END_REGION

REGION Network 129: Timer đếm thời gian Tip Bồn 1
   RUNG wire#powerrail
      Contact( "PLC1_Step_Bon1_Tip" )
      { S7_Templates := "time_type := Time" } "Timers_PLC1".Timer_Tip_Bon1.TON(pt := T#3S, et =>)
      Coil( "PLC1_Tip_Bon1_Auto_Done" )
   END_RUNG
   // the same network as SCL:
   "Timers_PLC1".Timer_Tip_Bon1.TON(IN := "PLC1_Step_Bon1_Tip", PT := T#3S);
   "PLC1_Tip_Bon1_Auto_Done" := "Timers_PLC1".Timer_Tip_Bon1.Q;
END_REGION

REGION Network 130: Timer đếm thời gian Tip Bồn 2
   RUNG wire#powerrail
      Contact( "PLC1_Step_Bon2_Tip" )
      { S7_Templates := "time_type := Time" } "Timers_PLC1".Timer_Tip_Bon2.TON(pt := T#3S, et =>)
      Coil( "PLC1_Tip_Bon2_Auto_Done" )
   END_RUNG
   // the same network as SCL:
   "Timers_PLC1".Timer_Tip_Bon2.TON(IN := "PLC1_Step_Bon2_Tip", PT := T#3S);
   "PLC1_Tip_Bon2_Auto_Done" := "Timers_PLC1".Timer_Tip_Bon2.Q;
END_REGION

REGION Network 131: Reset FQ Bồn 1 khi không dosing
   RUNG wire#powerrail
      I_Contact( "PLC1_Step_Bon1_Dosing" )
      { S7_GenerateENO := "TRUE" } Move(in := 0.0, out1 => "FQ3200_Bon1_HMI")
   END_RUNG
   // the same network as SCL:
   IF NOT "PLC1_Step_Bon1_Dosing" THEN "FQ3200_Bon1_HMI" := 0.0; END_IF;
END_REGION

REGION Network 132: Mở nước Bồn 1
   RUNG wire#powerrail
      Contact( "PLC1_Step_Bon1_Dosing" )
      S_Coil( "V3230_Nuoc_Bon1" )
   END_RUNG
   // the same network as SCL:
   IF "PLC1_Step_Bon1_Dosing" THEN "V3230_Nuoc_Bon1" := TRUE; END_IF;
END_REGION

REGION Network 133: CV nước Bồn 1 mở 100 phần trăm
   RUNG wire#powerrail
      Contact( "PLC1_Step_Bon1_Dosing" )
      { S7_GenerateENO := "TRUE" } Move(in := 100.0, out1 => "CV3201_Nuoc_Bon1")
   END_RUNG
   // the same network as SCL:
   IF "PLC1_Step_Bon1_Dosing" THEN "CV3201_Nuoc_Bon1" := 100.0; END_IF;
END_REGION

REGION Network 134: Đóng nước Bồn 1 sau dosing
   RUNG wire#powerrail
      I_Contact( "PLC1_Step_Bon1_Dosing" )
      R_Coil( "V3230_Nuoc_Bon1" )
   END_RUNG
   // the same network as SCL:
   IF NOT "PLC1_Step_Bon1_Dosing" THEN "V3230_Nuoc_Bon1" := FALSE; END_IF;
END_REGION

REGION Network 135: Đặt tốc độ khuấy Bồn 1
   RUNG wire#powerrail
      Contact( "PLC1_Step_Bon1_Khuay" )
      { S7_GenerateENO := "TRUE" } Move(in := "HMI_SP_PLC1_Toc_Do_Bon1", out1 => "AGTR3260_Toc_Do_AO")
   END_RUNG
   // the same network as SCL:
   IF "PLC1_Step_Bon1_Khuay" THEN "AGTR3260_Toc_Do_AO" := "HMI_SP_PLC1_Toc_Do_Bon1"; END_IF;
END_REGION

REGION Network 136: Timer đếm thời gian khuấy Bồn 1
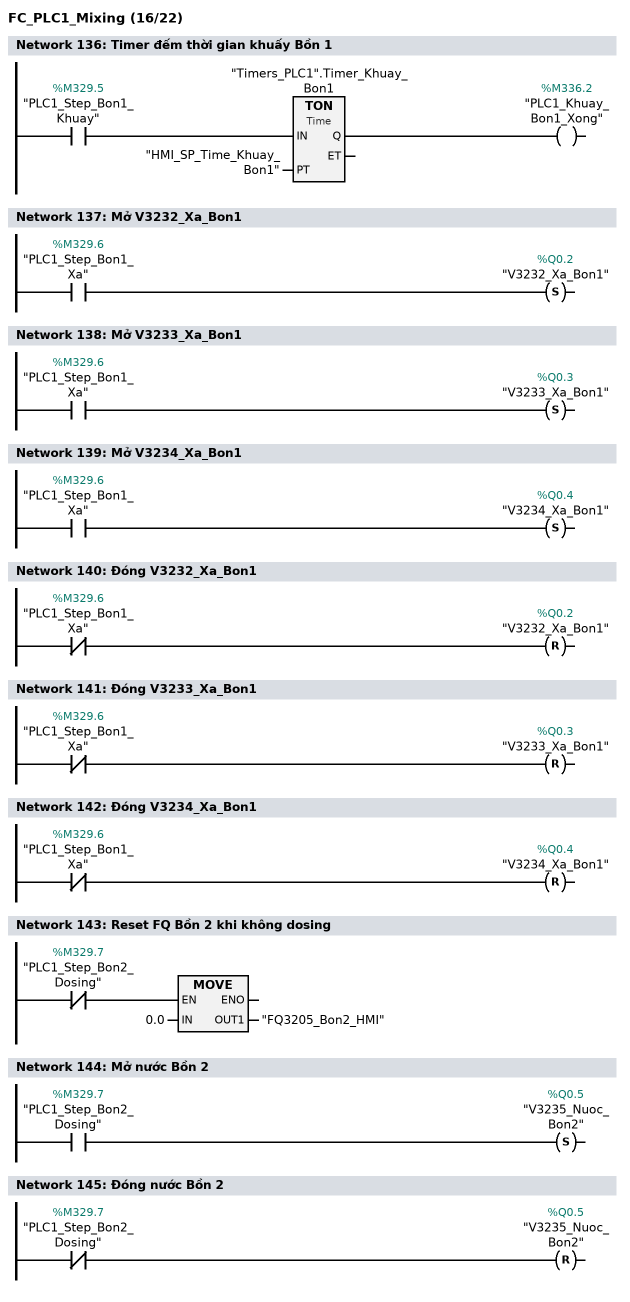
   RUNG wire#powerrail
      Contact( "PLC1_Step_Bon1_Khuay" )
      { S7_Templates := "time_type := Time" } "Timers_PLC1".Timer_Khuay_Bon1.TON(pt := "HMI_SP_Time_Khuay_Bon1", et =>)
      Coil( "PLC1_Khuay_Bon1_Xong" )
   END_RUNG
   // the same network as SCL:
   "Timers_PLC1".Timer_Khuay_Bon1.TON(IN := "PLC1_Step_Bon1_Khuay", PT := "HMI_SP_Time_Khuay_Bon1");
   "PLC1_Khuay_Bon1_Xong" := "Timers_PLC1".Timer_Khuay_Bon1.Q;
END_REGION

REGION Network 137: Mở V3232_Xa_Bon1
   RUNG wire#powerrail
      Contact( "PLC1_Step_Bon1_Xa" )
      S_Coil( "V3232_Xa_Bon1" )
   END_RUNG
   // the same network as SCL:
   IF "PLC1_Step_Bon1_Xa" THEN "V3232_Xa_Bon1" := TRUE; END_IF;
END_REGION

REGION Network 138: Mở V3233_Xa_Bon1
   RUNG wire#powerrail
      Contact( "PLC1_Step_Bon1_Xa" )
      S_Coil( "V3233_Xa_Bon1" )
   END_RUNG
   // the same network as SCL:
   IF "PLC1_Step_Bon1_Xa" THEN "V3233_Xa_Bon1" := TRUE; END_IF;
END_REGION

REGION Network 139: Mở V3234_Xa_Bon1
   RUNG wire#powerrail
      Contact( "PLC1_Step_Bon1_Xa" )
      S_Coil( "V3234_Xa_Bon1" )
   END_RUNG
   // the same network as SCL:
   IF "PLC1_Step_Bon1_Xa" THEN "V3234_Xa_Bon1" := TRUE; END_IF;
END_REGION

REGION Network 140: Đóng V3232_Xa_Bon1
   RUNG wire#powerrail
      I_Contact( "PLC1_Step_Bon1_Xa" )
      R_Coil( "V3232_Xa_Bon1" )
   END_RUNG
   // the same network as SCL:
   IF NOT "PLC1_Step_Bon1_Xa" THEN "V3232_Xa_Bon1" := FALSE; END_IF;
END_REGION

REGION Network 141: Đóng V3233_Xa_Bon1
   RUNG wire#powerrail
      I_Contact( "PLC1_Step_Bon1_Xa" )
      R_Coil( "V3233_Xa_Bon1" )
   END_RUNG
   // the same network as SCL:
   IF NOT "PLC1_Step_Bon1_Xa" THEN "V3233_Xa_Bon1" := FALSE; END_IF;
END_REGION

REGION Network 142: Đóng V3234_Xa_Bon1
   RUNG wire#powerrail
      I_Contact( "PLC1_Step_Bon1_Xa" )
      R_Coil( "V3234_Xa_Bon1" )
   END_RUNG
   // the same network as SCL:
   IF NOT "PLC1_Step_Bon1_Xa" THEN "V3234_Xa_Bon1" := FALSE; END_IF;
END_REGION

REGION Network 143: Reset FQ Bồn 2 khi không dosing
   RUNG wire#powerrail
      I_Contact( "PLC1_Step_Bon2_Dosing" )
      { S7_GenerateENO := "TRUE" } Move(in := 0.0, out1 => "FQ3205_Bon2_HMI")
   END_RUNG
   // the same network as SCL:
   IF NOT "PLC1_Step_Bon2_Dosing" THEN "FQ3205_Bon2_HMI" := 0.0; END_IF;
END_REGION

REGION Network 144: Mở nước Bồn 2
   RUNG wire#powerrail
      Contact( "PLC1_Step_Bon2_Dosing" )
      S_Coil( "V3235_Nuoc_Bon2" )
   END_RUNG
   // the same network as SCL:
   IF "PLC1_Step_Bon2_Dosing" THEN "V3235_Nuoc_Bon2" := TRUE; END_IF;
END_REGION

REGION Network 145: Đóng nước Bồn 2
   RUNG wire#powerrail
      I_Contact( "PLC1_Step_Bon2_Dosing" )
      R_Coil( "V3235_Nuoc_Bon2" )
   END_RUNG
   // the same network as SCL:
   IF NOT "PLC1_Step_Bon2_Dosing" THEN "V3235_Nuoc_Bon2" := FALSE; END_IF;
END_REGION

REGION Network 146: Tốc độ khuấy thuận Bồn 2
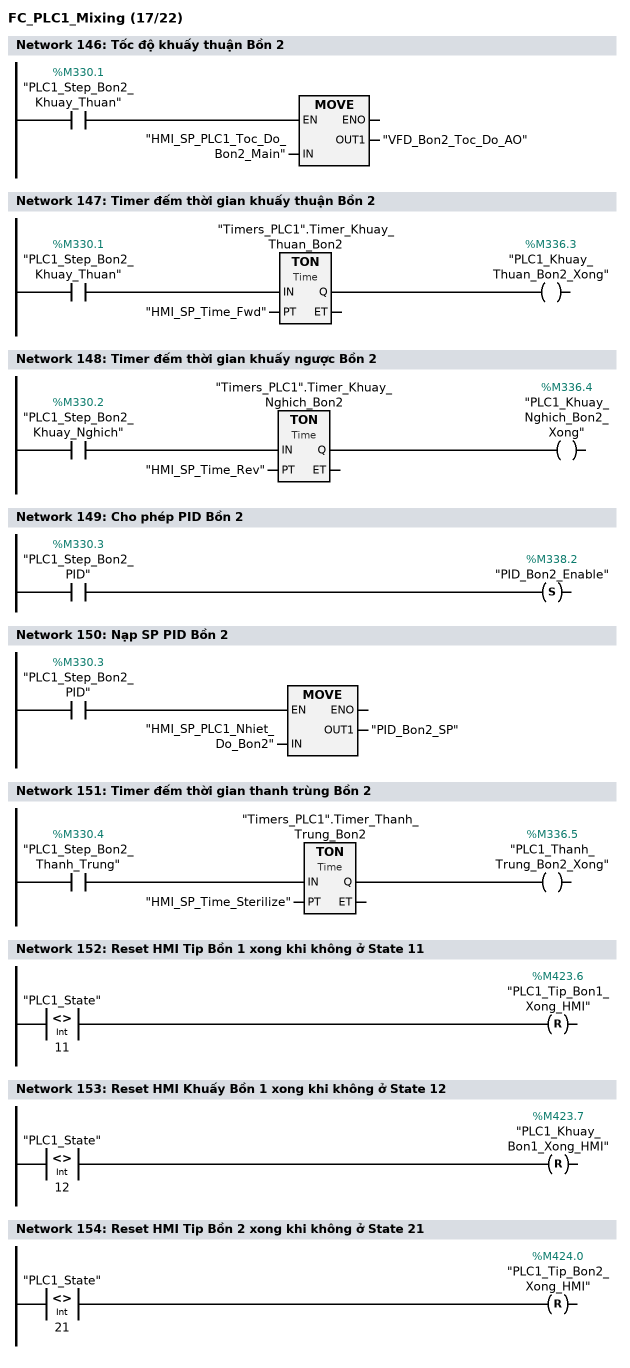
   RUNG wire#powerrail
      Contact( "PLC1_Step_Bon2_Khuay_Thuan" )
      { S7_GenerateENO := "TRUE" } Move(in := "HMI_SP_PLC1_Toc_Do_Bon2_Main", out1 => "VFD_Bon2_Toc_Do_AO")
   END_RUNG
   // the same network as SCL:
   IF "PLC1_Step_Bon2_Khuay_Thuan" THEN "VFD_Bon2_Toc_Do_AO" := "HMI_SP_PLC1_Toc_Do_Bon2_Main"; END_IF;
END_REGION

REGION Network 147: Timer đếm thời gian khuấy thuận Bồn 2
   RUNG wire#powerrail
      Contact( "PLC1_Step_Bon2_Khuay_Thuan" )
      { S7_Templates := "time_type := Time" } "Timers_PLC1".Timer_Khuay_Thuan_Bon2.TON(pt := "HMI_SP_Time_Fwd", et =>)
      Coil( "PLC1_Khuay_Thuan_Bon2_Xong" )
   END_RUNG
   // the same network as SCL:
   "Timers_PLC1".Timer_Khuay_Thuan_Bon2.TON(IN := "PLC1_Step_Bon2_Khuay_Thuan", PT := "HMI_SP_Time_Fwd");
   "PLC1_Khuay_Thuan_Bon2_Xong" := "Timers_PLC1".Timer_Khuay_Thuan_Bon2.Q;
END_REGION

REGION Network 148: Timer đếm thời gian khuấy ngược Bồn 2
   RUNG wire#powerrail
      Contact( "PLC1_Step_Bon2_Khuay_Nghich" )
      { S7_Templates := "time_type := Time" } "Timers_PLC1".Timer_Khuay_Nghich_Bon2.TON(pt := "HMI_SP_Time_Rev", et =>)
      Coil( "PLC1_Khuay_Nghich_Bon2_Xong" )
   END_RUNG
   // the same network as SCL:
   "Timers_PLC1".Timer_Khuay_Nghich_Bon2.TON(IN := "PLC1_Step_Bon2_Khuay_Nghich", PT := "HMI_SP_Time_Rev");
   "PLC1_Khuay_Nghich_Bon2_Xong" := "Timers_PLC1".Timer_Khuay_Nghich_Bon2.Q;
END_REGION

REGION Network 149: Cho phép PID Bồn 2
   RUNG wire#powerrail
      Contact( "PLC1_Step_Bon2_PID" )
      S_Coil( "PID_Bon2_Enable" )
   END_RUNG
   // the same network as SCL:
   IF "PLC1_Step_Bon2_PID" THEN "PID_Bon2_Enable" := TRUE; END_IF;
END_REGION

REGION Network 150: Nạp SP PID Bồn 2
   RUNG wire#powerrail
      Contact( "PLC1_Step_Bon2_PID" )
      { S7_GenerateENO := "TRUE" } Move(in := "HMI_SP_PLC1_Nhiet_Do_Bon2", out1 => "PID_Bon2_SP")
   END_RUNG
   // the same network as SCL:
   IF "PLC1_Step_Bon2_PID" THEN "PID_Bon2_SP" := "HMI_SP_PLC1_Nhiet_Do_Bon2"; END_IF;
END_REGION

REGION Network 151: Timer đếm thời gian thanh trùng Bồn 2
   RUNG wire#powerrail
      Contact( "PLC1_Step_Bon2_Thanh_Trung" )
      { S7_Templates := "time_type := Time" } "Timers_PLC1".Timer_Thanh_Trung_Bon2.TON(pt := "HMI_SP_Time_Sterilize", et =>)
      Coil( "PLC1_Thanh_Trung_Bon2_Xong" )
   END_RUNG
   // the same network as SCL:
   "Timers_PLC1".Timer_Thanh_Trung_Bon2.TON(IN := "PLC1_Step_Bon2_Thanh_Trung", PT := "HMI_SP_Time_Sterilize");
   "PLC1_Thanh_Trung_Bon2_Xong" := "Timers_PLC1".Timer_Thanh_Trung_Bon2.Q;
END_REGION

REGION Network 152: Reset HMI Tip Bồn 1 xong khi không ở State 11
   RUNG wire#powerrail
      { S7_Templates := "SrcType := Int" } NE_Contact(in1 := "PLC1_State", in2 := 11)
      R_Coil( "PLC1_Tip_Bon1_Xong_HMI" )
   END_RUNG
   // the same network as SCL:
   IF "PLC1_State" <> 11 THEN "PLC1_Tip_Bon1_Xong_HMI" := FALSE; END_IF;
END_REGION

REGION Network 153: Reset HMI Khuấy Bồn 1 xong khi không ở State 12
   RUNG wire#powerrail
      { S7_Templates := "SrcType := Int" } NE_Contact(in1 := "PLC1_State", in2 := 12)
      R_Coil( "PLC1_Khuay_Bon1_Xong_HMI" )
   END_RUNG
   // the same network as SCL:
   IF "PLC1_State" <> 12 THEN "PLC1_Khuay_Bon1_Xong_HMI" := FALSE; END_IF;
END_REGION

REGION Network 154: Reset HMI Tip Bồn 2 xong khi không ở State 21
   RUNG wire#powerrail
      { S7_Templates := "SrcType := Int" } NE_Contact(in1 := "PLC1_State", in2 := 21)
      R_Coil( "PLC1_Tip_Bon2_Xong_HMI" )
   END_RUNG
   // the same network as SCL:
   IF "PLC1_State" <> 21 THEN "PLC1_Tip_Bon2_Xong_HMI" := FALSE; END_IF;
END_REGION

REGION Network 155: Reset HMI Khuấy thuận Bồn 2 xong khi không ở State 22
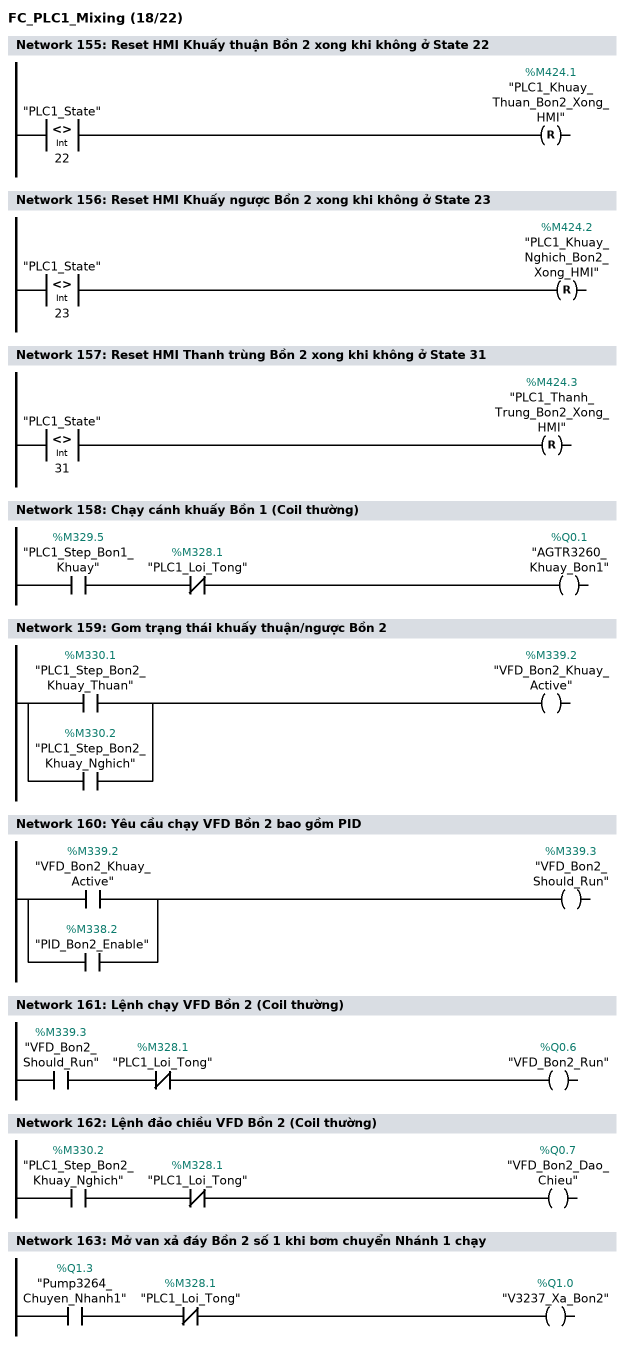
   RUNG wire#powerrail
      { S7_Templates := "SrcType := Int" } NE_Contact(in1 := "PLC1_State", in2 := 22)
      R_Coil( "PLC1_Khuay_Thuan_Bon2_Xong_HMI" )
   END_RUNG
   // the same network as SCL:
   IF "PLC1_State" <> 22 THEN "PLC1_Khuay_Thuan_Bon2_Xong_HMI" := FALSE; END_IF;
END_REGION

REGION Network 156: Reset HMI Khuấy ngược Bồn 2 xong khi không ở State 23
   RUNG wire#powerrail
      { S7_Templates := "SrcType := Int" } NE_Contact(in1 := "PLC1_State", in2 := 23)
      R_Coil( "PLC1_Khuay_Nghich_Bon2_Xong_HMI" )
   END_RUNG
   // the same network as SCL:
   IF "PLC1_State" <> 23 THEN "PLC1_Khuay_Nghich_Bon2_Xong_HMI" := FALSE; END_IF;
END_REGION

REGION Network 157: Reset HMI Thanh trùng Bồn 2 xong khi không ở State 31
   RUNG wire#powerrail
      { S7_Templates := "SrcType := Int" } NE_Contact(in1 := "PLC1_State", in2 := 31)
      R_Coil( "PLC1_Thanh_Trung_Bon2_Xong_HMI" )
   END_RUNG
   // the same network as SCL:
   IF "PLC1_State" <> 31 THEN "PLC1_Thanh_Trung_Bon2_Xong_HMI" := FALSE; END_IF;
END_REGION

REGION Network 158: Chạy cánh khuấy Bồn 1 (Coil thường)
   RUNG wire#powerrail
      Contact( "PLC1_Step_Bon1_Khuay" )
      I_Contact( "PLC1_Loi_Tong" )
      Coil( "AGTR3260_Khuay_Bon1" )
   END_RUNG
   // the same network as SCL:
   "AGTR3260_Khuay_Bon1" := "PLC1_Step_Bon1_Khuay" AND NOT "PLC1_Loi_Tong";
END_REGION

REGION Network 159: Gom trạng thái khuấy thuận/ngược Bồn 2
   RUNG wire#powerrail
      Contact( "PLC1_Step_Bon2_Khuay_Thuan" )
      wire#w1
      Coil( "VFD_Bon2_Khuay_Active" )
   END_RUNG
   RUNG wire#powerrail
      Contact( "PLC1_Step_Bon2_Khuay_Nghich" )
   END_RUNG wire#w1
   // the same network as SCL:
   "VFD_Bon2_Khuay_Active" := "PLC1_Step_Bon2_Khuay_Thuan" OR "PLC1_Step_Bon2_Khuay_Nghich";
END_REGION

REGION Network 160: Yêu cầu chạy VFD Bồn 2 bao gồm PID
   RUNG wire#powerrail
      Contact( "VFD_Bon2_Khuay_Active" )
      wire#w1
      Coil( "VFD_Bon2_Should_Run" )
   END_RUNG
   RUNG wire#powerrail
      Contact( "PID_Bon2_Enable" )
   END_RUNG wire#w1
   // the same network as SCL:
   "VFD_Bon2_Should_Run" := "VFD_Bon2_Khuay_Active" OR "PID_Bon2_Enable";
END_REGION

REGION Network 161: Lệnh chạy VFD Bồn 2 (Coil thường)
   RUNG wire#powerrail
      Contact( "VFD_Bon2_Should_Run" )
      I_Contact( "PLC1_Loi_Tong" )
      Coil( "VFD_Bon2_Run" )
   END_RUNG
   // the same network as SCL:
   "VFD_Bon2_Run" := "VFD_Bon2_Should_Run" AND NOT "PLC1_Loi_Tong";
END_REGION

REGION Network 162: Lệnh đảo chiều VFD Bồn 2 (Coil thường)
   RUNG wire#powerrail
      Contact( "PLC1_Step_Bon2_Khuay_Nghich" )
      I_Contact( "PLC1_Loi_Tong" )
      Coil( "VFD_Bon2_Dao_Chieu" )
   END_RUNG
   // the same network as SCL:
   "VFD_Bon2_Dao_Chieu" := "PLC1_Step_Bon2_Khuay_Nghich" AND NOT "PLC1_Loi_Tong";
END_REGION

REGION Network 163: Mở van xả đáy Bồn 2 số 1 khi bơm chuyển Nhánh 1 chạy
   RUNG wire#powerrail
      Contact( "Pump3264_Chuyen_Nhanh1" )
      I_Contact( "PLC1_Loi_Tong" )
      Coil( "V3237_Xa_Bon2" )
   END_RUNG
   // the same network as SCL:
   "V3237_Xa_Bon2" := "Pump3264_Chuyen_Nhanh1" AND NOT "PLC1_Loi_Tong";
END_REGION

REGION Network 164: Mở van xả đáy Bồn 2 số 2 khi bơm chuyển Nhánh 1 chạy
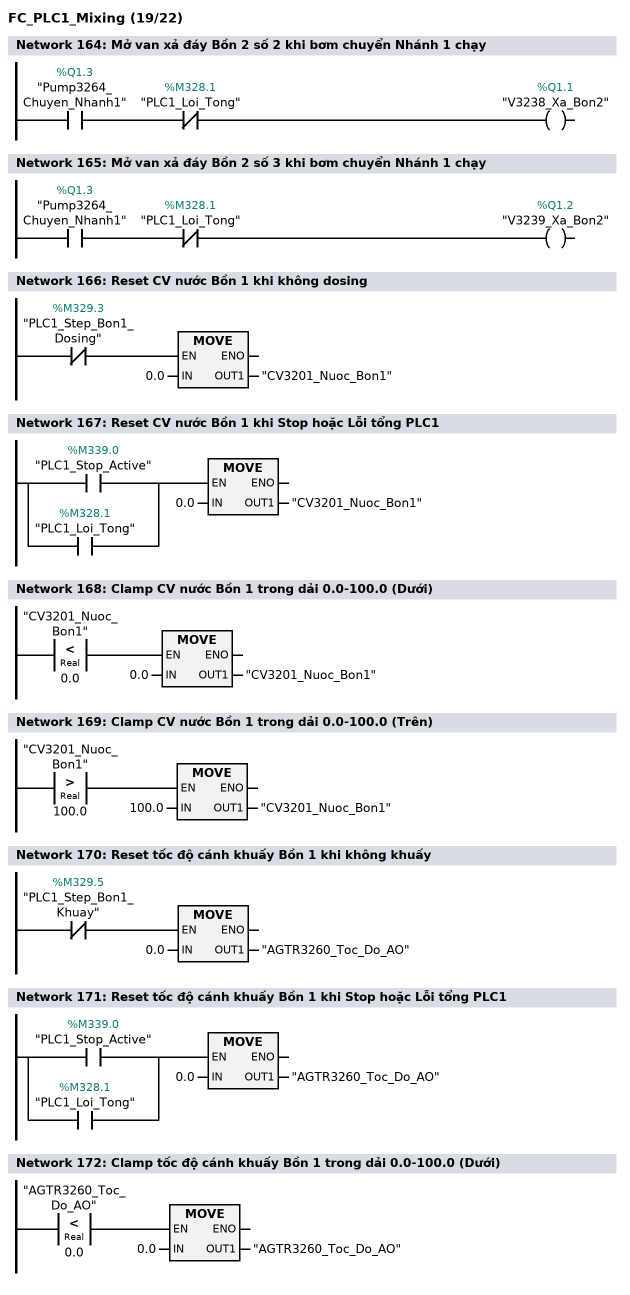
   RUNG wire#powerrail
      Contact( "Pump3264_Chuyen_Nhanh1" )
      I_Contact( "PLC1_Loi_Tong" )
      Coil( "V3238_Xa_Bon2" )
   END_RUNG
   // the same network as SCL:
   "V3238_Xa_Bon2" := "Pump3264_Chuyen_Nhanh1" AND NOT "PLC1_Loi_Tong";
END_REGION

REGION Network 165: Mở van xả đáy Bồn 2 số 3 khi bơm chuyển Nhánh 1 chạy
   RUNG wire#powerrail
      Contact( "Pump3264_Chuyen_Nhanh1" )
      I_Contact( "PLC1_Loi_Tong" )
      Coil( "V3239_Xa_Bon2" )
   END_RUNG
   // the same network as SCL:
   "V3239_Xa_Bon2" := "Pump3264_Chuyen_Nhanh1" AND NOT "PLC1_Loi_Tong";
END_REGION

REGION Network 166: Reset CV nước Bồn 1 khi không dosing
   RUNG wire#powerrail
      I_Contact( "PLC1_Step_Bon1_Dosing" )
      { S7_GenerateENO := "TRUE" } Move(in := 0.0, out1 => "CV3201_Nuoc_Bon1")
   END_RUNG
   // the same network as SCL:
   IF NOT "PLC1_Step_Bon1_Dosing" THEN "CV3201_Nuoc_Bon1" := 0.0; END_IF;
END_REGION

REGION Network 167: Reset CV nước Bồn 1 khi Stop hoặc Lỗi tổng PLC1
   RUNG wire#powerrail
      Contact( "PLC1_Stop_Active" )
      wire#w1
      { S7_GenerateENO := "TRUE" } Move(in := 0.0, out1 => "CV3201_Nuoc_Bon1")
   END_RUNG
   RUNG wire#powerrail
      Contact( "PLC1_Loi_Tong" )
   END_RUNG wire#w1
   // the same network as SCL:
   IF "PLC1_Stop_Active" OR "PLC1_Loi_Tong" THEN "CV3201_Nuoc_Bon1" := 0.0; END_IF;
END_REGION

REGION Network 168: Clamp CV nước Bồn 1 trong dải 0.0-100.0 (Dưới)
   RUNG wire#powerrail
      { S7_Templates := "SrcType := Real" } LT_Contact(in1 := "CV3201_Nuoc_Bon1", in2 := 0.0)
      { S7_GenerateENO := "TRUE" } Move(in := 0.0, out1 => "CV3201_Nuoc_Bon1")
   END_RUNG
   // the same network as SCL:
   IF "CV3201_Nuoc_Bon1" < 0.0 THEN "CV3201_Nuoc_Bon1" := 0.0; END_IF;
END_REGION

REGION Network 169: Clamp CV nước Bồn 1 trong dải 0.0-100.0 (Trên)
   RUNG wire#powerrail
      { S7_Templates := "SrcType := Real" } GT_Contact(in1 := "CV3201_Nuoc_Bon1", in2 := 100.0)
      { S7_GenerateENO := "TRUE" } Move(in := 100.0, out1 => "CV3201_Nuoc_Bon1")
   END_RUNG
   // the same network as SCL:
   IF "CV3201_Nuoc_Bon1" > 100.0 THEN "CV3201_Nuoc_Bon1" := 100.0; END_IF;
END_REGION

REGION Network 170: Reset tốc độ cánh khuấy Bồn 1 khi không khuấy
   RUNG wire#powerrail
      I_Contact( "PLC1_Step_Bon1_Khuay" )
      { S7_GenerateENO := "TRUE" } Move(in := 0.0, out1 => "AGTR3260_Toc_Do_AO")
   END_RUNG
   // the same network as SCL:
   IF NOT "PLC1_Step_Bon1_Khuay" THEN "AGTR3260_Toc_Do_AO" := 0.0; END_IF;
END_REGION

REGION Network 171: Reset tốc độ cánh khuấy Bồn 1 khi Stop hoặc Lỗi tổng PLC1
   RUNG wire#powerrail
      Contact( "PLC1_Stop_Active" )
      wire#w1
      { S7_GenerateENO := "TRUE" } Move(in := 0.0, out1 => "AGTR3260_Toc_Do_AO")
   END_RUNG
   RUNG wire#powerrail
      Contact( "PLC1_Loi_Tong" )
   END_RUNG wire#w1
   // the same network as SCL:
   IF "PLC1_Stop_Active" OR "PLC1_Loi_Tong" THEN "AGTR3260_Toc_Do_AO" := 0.0; END_IF;
END_REGION

REGION Network 172: Clamp tốc độ cánh khuấy Bồn 1 trong dải 0.0-100.0 (Dưới)
   RUNG wire#powerrail
      { S7_Templates := "SrcType := Real" } LT_Contact(in1 := "AGTR3260_Toc_Do_AO", in2 := 0.0)
      { S7_GenerateENO := "TRUE" } Move(in := 0.0, out1 => "AGTR3260_Toc_Do_AO")
   END_RUNG
   // the same network as SCL:
   IF "AGTR3260_Toc_Do_AO" < 0.0 THEN "AGTR3260_Toc_Do_AO" := 0.0; END_IF;
END_REGION

REGION Network 173: Clamp tốc độ cánh khuấy Bồn 1 trong dải 0.0-100.0 (Trên)
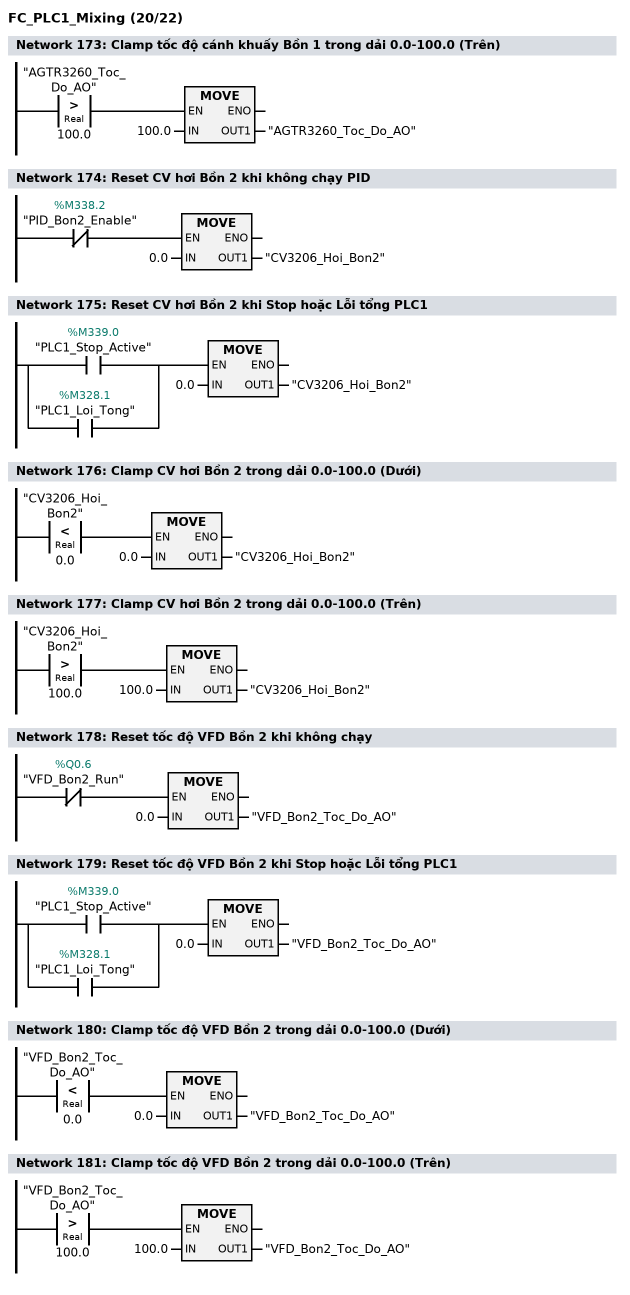
   RUNG wire#powerrail
      { S7_Templates := "SrcType := Real" } GT_Contact(in1 := "AGTR3260_Toc_Do_AO", in2 := 100.0)
      { S7_GenerateENO := "TRUE" } Move(in := 100.0, out1 => "AGTR3260_Toc_Do_AO")
   END_RUNG
   // the same network as SCL:
   IF "AGTR3260_Toc_Do_AO" > 100.0 THEN "AGTR3260_Toc_Do_AO" := 100.0; END_IF;
END_REGION

REGION Network 174: Reset CV hơi Bồn 2 khi không chạy PID
   RUNG wire#powerrail
      I_Contact( "PID_Bon2_Enable" )
      { S7_GenerateENO := "TRUE" } Move(in := 0.0, out1 => "CV3206_Hoi_Bon2")
   END_RUNG
   // the same network as SCL:
   IF NOT "PID_Bon2_Enable" THEN "CV3206_Hoi_Bon2" := 0.0; END_IF;
END_REGION

REGION Network 175: Reset CV hơi Bồn 2 khi Stop hoặc Lỗi tổng PLC1
   RUNG wire#powerrail
      Contact( "PLC1_Stop_Active" )
      wire#w1
      { S7_GenerateENO := "TRUE" } Move(in := 0.0, out1 => "CV3206_Hoi_Bon2")
   END_RUNG
   RUNG wire#powerrail
      Contact( "PLC1_Loi_Tong" )
   END_RUNG wire#w1
   // the same network as SCL:
   IF "PLC1_Stop_Active" OR "PLC1_Loi_Tong" THEN "CV3206_Hoi_Bon2" := 0.0; END_IF;
END_REGION

REGION Network 176: Clamp CV hơi Bồn 2 trong dải 0.0-100.0 (Dưới)
   RUNG wire#powerrail
      { S7_Templates := "SrcType := Real" } LT_Contact(in1 := "CV3206_Hoi_Bon2", in2 := 0.0)
      { S7_GenerateENO := "TRUE" } Move(in := 0.0, out1 => "CV3206_Hoi_Bon2")
   END_RUNG
   // the same network as SCL:
   IF "CV3206_Hoi_Bon2" < 0.0 THEN "CV3206_Hoi_Bon2" := 0.0; END_IF;
END_REGION

REGION Network 177: Clamp CV hơi Bồn 2 trong dải 0.0-100.0 (Trên)
   RUNG wire#powerrail
      { S7_Templates := "SrcType := Real" } GT_Contact(in1 := "CV3206_Hoi_Bon2", in2 := 100.0)
      { S7_GenerateENO := "TRUE" } Move(in := 100.0, out1 => "CV3206_Hoi_Bon2")
   END_RUNG
   // the same network as SCL:
   IF "CV3206_Hoi_Bon2" > 100.0 THEN "CV3206_Hoi_Bon2" := 100.0; END_IF;
END_REGION

REGION Network 178: Reset tốc độ VFD Bồn 2 khi không chạy
   RUNG wire#powerrail
      I_Contact( "VFD_Bon2_Run" )
      { S7_GenerateENO := "TRUE" } Move(in := 0.0, out1 => "VFD_Bon2_Toc_Do_AO")
   END_RUNG
   // the same network as SCL:
   IF NOT "VFD_Bon2_Run" THEN "VFD_Bon2_Toc_Do_AO" := 0.0; END_IF;
END_REGION

REGION Network 179: Reset tốc độ VFD Bồn 2 khi Stop hoặc Lỗi tổng PLC1
   RUNG wire#powerrail
      Contact( "PLC1_Stop_Active" )
      wire#w1
      { S7_GenerateENO := "TRUE" } Move(in := 0.0, out1 => "VFD_Bon2_Toc_Do_AO")
   END_RUNG
   RUNG wire#powerrail
      Contact( "PLC1_Loi_Tong" )
   END_RUNG wire#w1
   // the same network as SCL:
   IF "PLC1_Stop_Active" OR "PLC1_Loi_Tong" THEN "VFD_Bon2_Toc_Do_AO" := 0.0; END_IF;
END_REGION

REGION Network 180: Clamp tốc độ VFD Bồn 2 trong dải 0.0-100.0 (Dưới)
   RUNG wire#powerrail
      { S7_Templates := "SrcType := Real" } LT_Contact(in1 := "VFD_Bon2_Toc_Do_AO", in2 := 0.0)
      { S7_GenerateENO := "TRUE" } Move(in := 0.0, out1 => "VFD_Bon2_Toc_Do_AO")
   END_RUNG
   // the same network as SCL:
   IF "VFD_Bon2_Toc_Do_AO" < 0.0 THEN "VFD_Bon2_Toc_Do_AO" := 0.0; END_IF;
END_REGION

REGION Network 181: Clamp tốc độ VFD Bồn 2 trong dải 0.0-100.0 (Trên)
   RUNG wire#powerrail
      { S7_Templates := "SrcType := Real" } GT_Contact(in1 := "VFD_Bon2_Toc_Do_AO", in2 := 100.0)
      { S7_GenerateENO := "TRUE" } Move(in := 100.0, out1 => "VFD_Bon2_Toc_Do_AO")
   END_RUNG
   // the same network as SCL:
   IF "VFD_Bon2_Toc_Do_AO" > 100.0 THEN "VFD_Bon2_Toc_Do_AO" := 100.0; END_IF;
END_REGION

REGION Network 182: VFD Bon 2 Freq Scale: Speed SP x 5.0
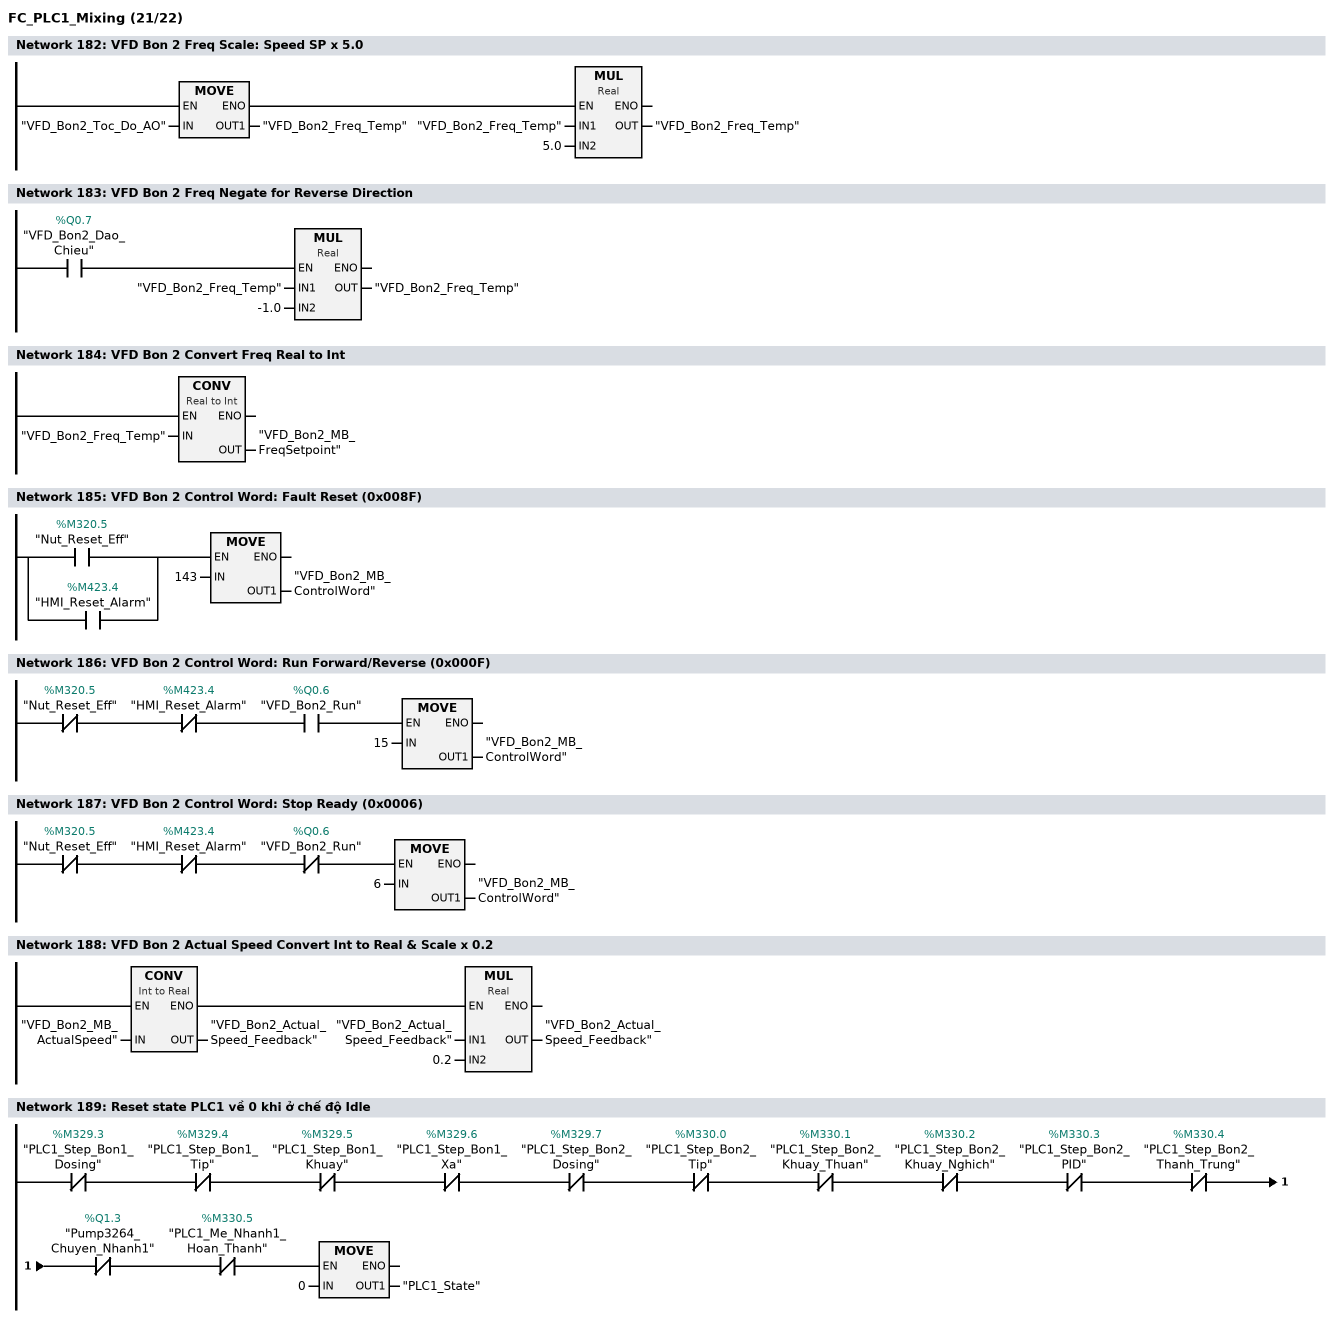
   RUNG wire#powerrail
      { S7_GenerateENO := "TRUE" } Move(in := "VFD_Bon2_Toc_Do_AO", out1 => "VFD_Bon2_Freq_Temp")
      { S7_Templates := "SrcType := Real"; S7_GenerateENO := "TRUE" } Mul(in1 := "VFD_Bon2_Freq_Temp", in2 := 5.0, out => "VFD_Bon2_Freq_Temp")
   END_RUNG
   // the same network as SCL:
   // ENO of a box is taken as its EN; it also drops when the box reports an error
   "VFD_Bon2_Freq_Temp" := "VFD_Bon2_Toc_Do_AO";
   "VFD_Bon2_Freq_Temp" := "VFD_Bon2_Freq_Temp" * 5.0;
END_REGION

REGION Network 183: VFD Bon 2 Freq Negate for Reverse Direction
   RUNG wire#powerrail
      Contact( "VFD_Bon2_Dao_Chieu" )
      { S7_Templates := "SrcType := Real"; S7_GenerateENO := "TRUE" } Mul(in1 := "VFD_Bon2_Freq_Temp", in2 := -1.0, out => "VFD_Bon2_Freq_Temp")
   END_RUNG
   // the same network as SCL:
   IF "VFD_Bon2_Dao_Chieu" THEN "VFD_Bon2_Freq_Temp" := "VFD_Bon2_Freq_Temp" * (-1.0); END_IF;
END_REGION

REGION Network 184: VFD Bon 2 Convert Freq Real to Int
   RUNG wire#powerrail
      { S7_Templates := "[SrcType := Real, DestType := Int]"; S7_GenerateENO := "TRUE" } Convert(in := "VFD_Bon2_Freq_Temp", out => "VFD_Bon2_MB_FreqSetpoint")
   END_RUNG
   // the same network as SCL:
   "VFD_Bon2_MB_FreqSetpoint" := REAL_TO_INT("VFD_Bon2_Freq_Temp");
END_REGION

REGION Network 185: VFD Bon 2 Control Word: Fault Reset (0x008F)
   RUNG wire#powerrail
      Contact( "Nut_Reset_Eff" )
      wire#w1
      { S7_GenerateENO := "TRUE" } Move(in := 143, out1 => "VFD_Bon2_MB_ControlWord")
   END_RUNG
   RUNG wire#powerrail
      Contact( "HMI_Reset_Alarm" )
   END_RUNG wire#w1
   // the same network as SCL:
   IF "Nut_Reset_Eff" OR "HMI_Reset_Alarm" THEN "VFD_Bon2_MB_ControlWord" := 143; END_IF;
END_REGION

REGION Network 186: VFD Bon 2 Control Word: Run Forward/Reverse (0x000F)
   RUNG wire#powerrail
      I_Contact( "Nut_Reset_Eff" )
      I_Contact( "HMI_Reset_Alarm" )
      Contact( "VFD_Bon2_Run" )
      { S7_GenerateENO := "TRUE" } Move(in := 15, out1 => "VFD_Bon2_MB_ControlWord")
   END_RUNG
   // the same network as SCL:
   IF NOT "Nut_Reset_Eff" AND NOT "HMI_Reset_Alarm" AND "VFD_Bon2_Run" THEN
       "VFD_Bon2_MB_ControlWord" := 15;
   END_IF;
END_REGION

REGION Network 187: VFD Bon 2 Control Word: Stop Ready (0x0006)
   RUNG wire#powerrail
      I_Contact( "Nut_Reset_Eff" )
      I_Contact( "HMI_Reset_Alarm" )
      I_Contact( "VFD_Bon2_Run" )
      { S7_GenerateENO := "TRUE" } Move(in := 6, out1 => "VFD_Bon2_MB_ControlWord")
   END_RUNG
   // the same network as SCL:
   IF NOT "Nut_Reset_Eff" AND NOT "HMI_Reset_Alarm" AND NOT "VFD_Bon2_Run" THEN
       "VFD_Bon2_MB_ControlWord" := 6;
   END_IF;
END_REGION

REGION Network 188: VFD Bon 2 Actual Speed Convert Int to Real & Scale x 0.2
   RUNG wire#powerrail
      { S7_Templates := "[SrcType := Int, DestType := Real]"; S7_GenerateENO := "TRUE" } Convert(in := "VFD_Bon2_MB_ActualSpeed", out => "VFD_Bon2_Actual_Speed_Feedback")
      { S7_Templates := "SrcType := Real"; S7_GenerateENO := "TRUE" } Mul(in1 := "VFD_Bon2_Actual_Speed_Feedback", in2 := 0.2, out => "VFD_Bon2_Actual_Speed_Feedback")
   END_RUNG
   // the same network as SCL:
   // ENO of a box is taken as its EN; it also drops when the box reports an error
   "VFD_Bon2_Actual_Speed_Feedback" := INT_TO_REAL("VFD_Bon2_MB_ActualSpeed");
   "VFD_Bon2_Actual_Speed_Feedback" := "VFD_Bon2_Actual_Speed_Feedback" * 0.2;
END_REGION

REGION Network 189: Reset state PLC1 về 0 khi ở chế độ Idle
   RUNG wire#powerrail
      I_Contact( "PLC1_Step_Bon1_Dosing" )
      I_Contact( "PLC1_Step_Bon1_Tip" )
      I_Contact( "PLC1_Step_Bon1_Khuay" )
      I_Contact( "PLC1_Step_Bon1_Xa" )
      I_Contact( "PLC1_Step_Bon2_Dosing" )
      I_Contact( "PLC1_Step_Bon2_Tip" )
      I_Contact( "PLC1_Step_Bon2_Khuay_Thuan" )
      I_Contact( "PLC1_Step_Bon2_Khuay_Nghich" )
      I_Contact( "PLC1_Step_Bon2_PID" )
      I_Contact( "PLC1_Step_Bon2_Thanh_Trung" )
      I_Contact( "Pump3264_Chuyen_Nhanh1" )
      I_Contact( "PLC1_Me_Nhanh1_Hoan_Thanh" )
      { S7_GenerateENO := "TRUE" } Move(in := 0, out1 => "PLC1_State")
   END_RUNG
   // the same network as SCL:
   IF NOT "PLC1_Step_Bon1_Dosing" AND NOT "PLC1_Step_Bon1_Tip" AND NOT "PLC1_Step_Bon1_Khuay" AND NOT "PLC1_Step_Bon1_Xa" AND NOT "PLC1_Step_Bon2_Dosing" AND NOT "PLC1_Step_Bon2_Tip" AND NOT "PLC1_Step_Bon2_Khuay_Thuan" AND NOT "PLC1_Step_Bon2_Khuay_Nghich" AND NOT "PLC1_Step_Bon2_PID" AND NOT "PLC1_Step_Bon2_Thanh_Trung" AND NOT "Pump3264_Chuyen_Nhanh1" AND NOT "PLC1_Me_Nhanh1_Hoan_Thanh" THEN
       "PLC1_State" := 0;
   END_IF;
END_REGION

REGION Network 190: Dừng an toàn PLC1 reset V3230_Nuoc_Bon1
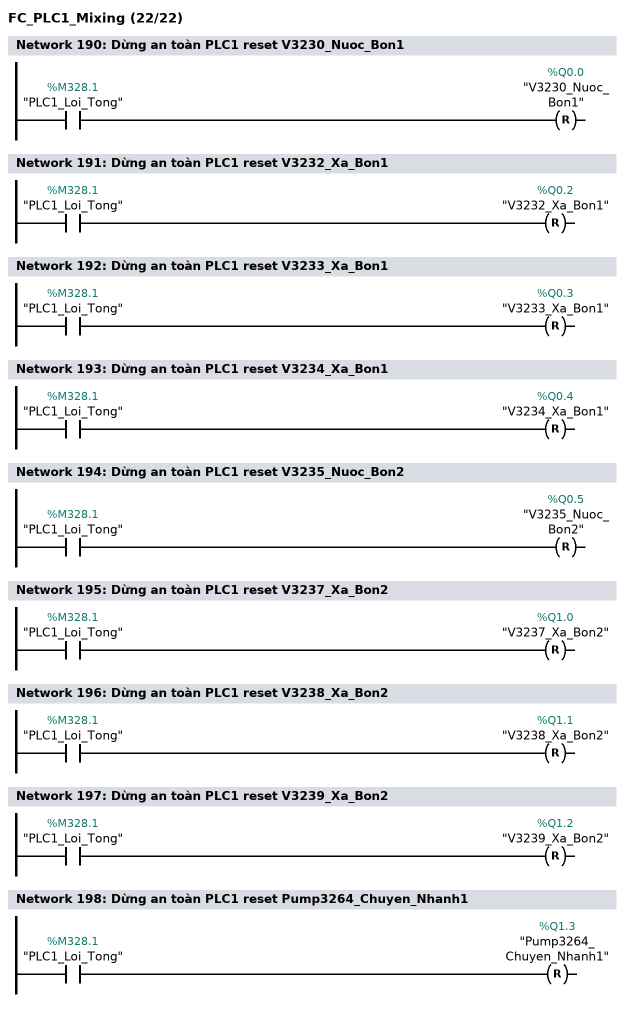
   RUNG wire#powerrail
      Contact( "PLC1_Loi_Tong" )
      R_Coil( "V3230_Nuoc_Bon1" )
   END_RUNG
   // the same network as SCL:
   IF "PLC1_Loi_Tong" THEN "V3230_Nuoc_Bon1" := FALSE; END_IF;
END_REGION

REGION Network 191: Dừng an toàn PLC1 reset V3232_Xa_Bon1
   RUNG wire#powerrail
      Contact( "PLC1_Loi_Tong" )
      R_Coil( "V3232_Xa_Bon1" )
   END_RUNG
   // the same network as SCL:
   IF "PLC1_Loi_Tong" THEN "V3232_Xa_Bon1" := FALSE; END_IF;
END_REGION

REGION Network 192: Dừng an toàn PLC1 reset V3233_Xa_Bon1
   RUNG wire#powerrail
      Contact( "PLC1_Loi_Tong" )
      R_Coil( "V3233_Xa_Bon1" )
   END_RUNG
   // the same network as SCL:
   IF "PLC1_Loi_Tong" THEN "V3233_Xa_Bon1" := FALSE; END_IF;
END_REGION

REGION Network 193: Dừng an toàn PLC1 reset V3234_Xa_Bon1
   RUNG wire#powerrail
      Contact( "PLC1_Loi_Tong" )
      R_Coil( "V3234_Xa_Bon1" )
   END_RUNG
   // the same network as SCL:
   IF "PLC1_Loi_Tong" THEN "V3234_Xa_Bon1" := FALSE; END_IF;
END_REGION

REGION Network 194: Dừng an toàn PLC1 reset V3235_Nuoc_Bon2
   RUNG wire#powerrail
      Contact( "PLC1_Loi_Tong" )
      R_Coil( "V3235_Nuoc_Bon2" )
   END_RUNG
   // the same network as SCL:
   IF "PLC1_Loi_Tong" THEN "V3235_Nuoc_Bon2" := FALSE; END_IF;
END_REGION

REGION Network 195: Dừng an toàn PLC1 reset V3237_Xa_Bon2
   RUNG wire#powerrail
      Contact( "PLC1_Loi_Tong" )
      R_Coil( "V3237_Xa_Bon2" )
   END_RUNG
   // the same network as SCL:
   IF "PLC1_Loi_Tong" THEN "V3237_Xa_Bon2" := FALSE; END_IF;
END_REGION

REGION Network 196: Dừng an toàn PLC1 reset V3238_Xa_Bon2
   RUNG wire#powerrail
      Contact( "PLC1_Loi_Tong" )
      R_Coil( "V3238_Xa_Bon2" )
   END_RUNG
   // the same network as SCL:
   IF "PLC1_Loi_Tong" THEN "V3238_Xa_Bon2" := FALSE; END_IF;
END_REGION

REGION Network 197: Dừng an toàn PLC1 reset V3239_Xa_Bon2
   RUNG wire#powerrail
      Contact( "PLC1_Loi_Tong" )
      R_Coil( "V3239_Xa_Bon2" )
   END_RUNG
   // the same network as SCL:
   IF "PLC1_Loi_Tong" THEN "V3239_Xa_Bon2" := FALSE; END_IF;
END_REGION

REGION Network 198: Dừng an toàn PLC1 reset Pump3264_Chuyen_Nhanh1
   RUNG wire#powerrail
      Contact( "PLC1_Loi_Tong" )
      R_Coil( "Pump3264_Chuyen_Nhanh1" )
   END_RUNG
   // the same network as SCL:
   IF "PLC1_Loi_Tong" THEN "Pump3264_Chuyen_Nhanh1" := FALSE; END_IF;
END_REGION
END_FUNCTION

FUNCTION "FC_Bon_Chua_Loc" : Void   // FC30, LAD
{ S7_Optimized_Access := 'TRUE' }
VERSION : 0.1
// stored: AutoNumber true, IsIECCheckEnabled false, SetENOAutomatically false, UDAEnableTagReadback false
   VAR_TEMP   // added for the SCL form of the ladder/FBD networks
      _w1 : Bool;
   END_VAR
BEGIN

REGION Network 1: Gated HMI LSH3310_Pheu_Cao qua Sim Mode
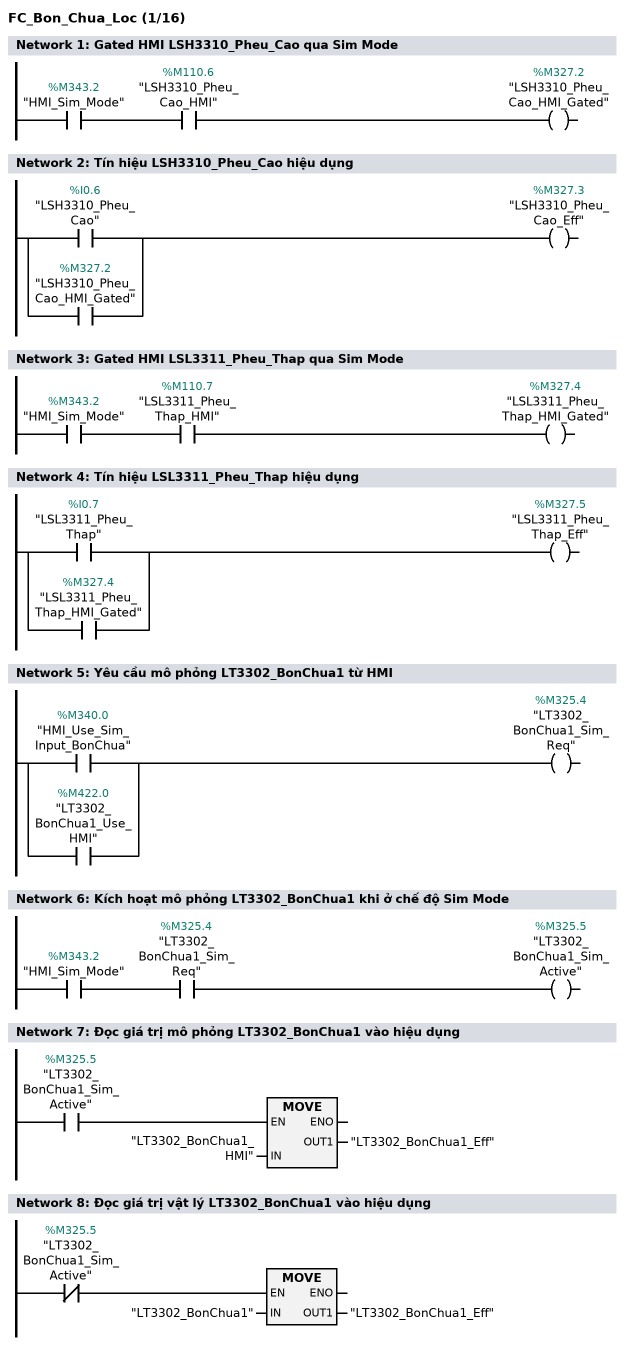
   RUNG wire#powerrail
      Contact( "HMI_Sim_Mode" )
      Contact( "LSH3310_Pheu_Cao_HMI" )
      Coil( "LSH3310_Pheu_Cao_HMI_Gated" )
   END_RUNG
   // the same network as SCL:
   "LSH3310_Pheu_Cao_HMI_Gated" := "HMI_Sim_Mode" AND "LSH3310_Pheu_Cao_HMI";
END_REGION

REGION Network 2: Tín hiệu LSH3310_Pheu_Cao hiệu dụng
   RUNG wire#powerrail
      Contact( "LSH3310_Pheu_Cao" )
      wire#w1
      Coil( "LSH3310_Pheu_Cao_Eff" )
   END_RUNG
   RUNG wire#powerrail
      Contact( "LSH3310_Pheu_Cao_HMI_Gated" )
   END_RUNG wire#w1
   // the same network as SCL:
   "LSH3310_Pheu_Cao_Eff" := "LSH3310_Pheu_Cao" OR "LSH3310_Pheu_Cao_HMI_Gated";
END_REGION

REGION Network 3: Gated HMI LSL3311_Pheu_Thap qua Sim Mode
   RUNG wire#powerrail
      Contact( "HMI_Sim_Mode" )
      Contact( "LSL3311_Pheu_Thap_HMI" )
      Coil( "LSL3311_Pheu_Thap_HMI_Gated" )
   END_RUNG
   // the same network as SCL:
   "LSL3311_Pheu_Thap_HMI_Gated" := "HMI_Sim_Mode" AND "LSL3311_Pheu_Thap_HMI";
END_REGION

REGION Network 4: Tín hiệu LSL3311_Pheu_Thap hiệu dụng
   RUNG wire#powerrail
      Contact( "LSL3311_Pheu_Thap" )
      wire#w1
      Coil( "LSL3311_Pheu_Thap_Eff" )
   END_RUNG
   RUNG wire#powerrail
      Contact( "LSL3311_Pheu_Thap_HMI_Gated" )
   END_RUNG wire#w1
   // the same network as SCL:
   "LSL3311_Pheu_Thap_Eff" := "LSL3311_Pheu_Thap" OR "LSL3311_Pheu_Thap_HMI_Gated";
END_REGION

REGION Network 5: Yêu cầu mô phỏng LT3302_BonChua1 từ HMI
   RUNG wire#powerrail
      Contact( "HMI_Use_Sim_Input_BonChua" )
      wire#w1
      Coil( "LT3302_BonChua1_Sim_Req" )
   END_RUNG
   RUNG wire#powerrail
      Contact( "LT3302_BonChua1_Use_HMI" )
   END_RUNG wire#w1
   // the same network as SCL:
   "LT3302_BonChua1_Sim_Req" := "HMI_Use_Sim_Input_BonChua" OR "LT3302_BonChua1_Use_HMI";
END_REGION

REGION Network 6: Kích hoạt mô phỏng LT3302_BonChua1 khi ở chế độ Sim Mode
   RUNG wire#powerrail
      Contact( "HMI_Sim_Mode" )
      Contact( "LT3302_BonChua1_Sim_Req" )
      Coil( "LT3302_BonChua1_Sim_Active" )
   END_RUNG
   // the same network as SCL:
   "LT3302_BonChua1_Sim_Active" := "HMI_Sim_Mode" AND "LT3302_BonChua1_Sim_Req";
END_REGION

REGION Network 7: Đọc giá trị mô phỏng LT3302_BonChua1 vào hiệu dụng
   RUNG wire#powerrail
      Contact( "LT3302_BonChua1_Sim_Active" )
      { S7_GenerateENO := "TRUE" } Move(in := "LT3302_BonChua1_HMI", out1 => "LT3302_BonChua1_Eff")
   END_RUNG
   // the same network as SCL:
   IF "LT3302_BonChua1_Sim_Active" THEN "LT3302_BonChua1_Eff" := "LT3302_BonChua1_HMI"; END_IF;
END_REGION

REGION Network 8: Đọc giá trị vật lý LT3302_BonChua1 vào hiệu dụng
   RUNG wire#powerrail
      I_Contact( "LT3302_BonChua1_Sim_Active" )
      { S7_GenerateENO := "TRUE" } Move(in := "LT3302_BonChua1", out1 => "LT3302_BonChua1_Eff")
   END_RUNG
   // the same network as SCL:
   IF NOT "LT3302_BonChua1_Sim_Active" THEN "LT3302_BonChua1_Eff" := "LT3302_BonChua1"; END_IF;
END_REGION

REGION Network 9: Yêu cầu mô phỏng TT3301_BonChua1 từ HMI
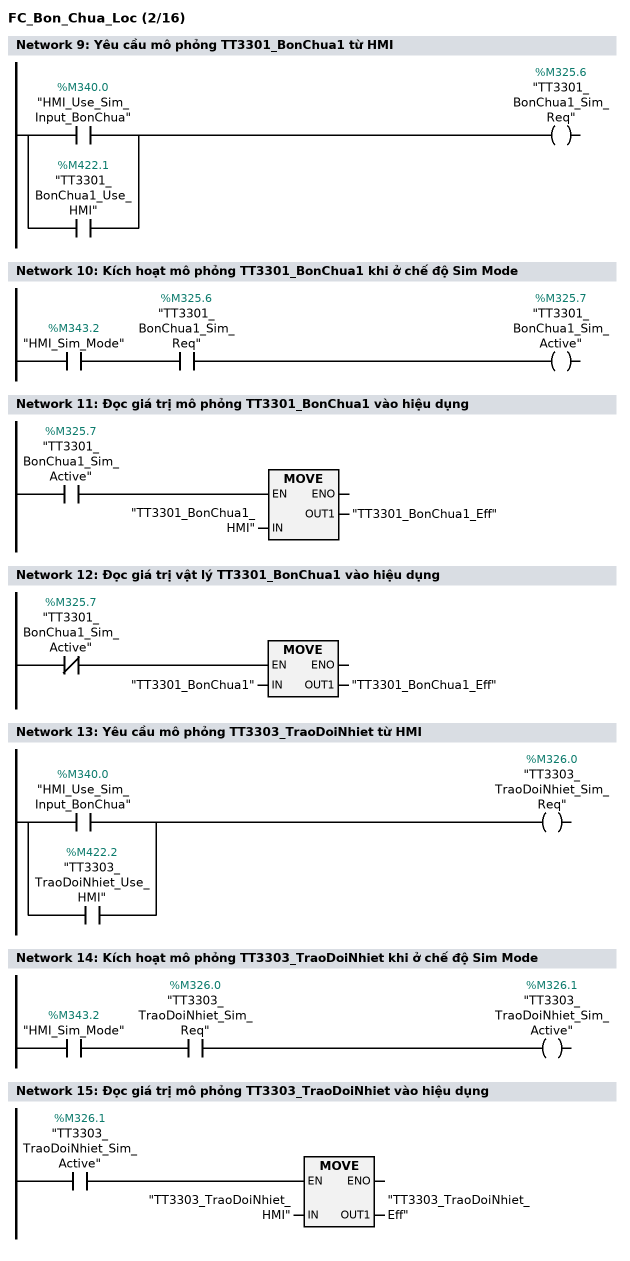
   RUNG wire#powerrail
      Contact( "HMI_Use_Sim_Input_BonChua" )
      wire#w1
      Coil( "TT3301_BonChua1_Sim_Req" )
   END_RUNG
   RUNG wire#powerrail
      Contact( "TT3301_BonChua1_Use_HMI" )
   END_RUNG wire#w1
   // the same network as SCL:
   "TT3301_BonChua1_Sim_Req" := "HMI_Use_Sim_Input_BonChua" OR "TT3301_BonChua1_Use_HMI";
END_REGION

REGION Network 10: Kích hoạt mô phỏng TT3301_BonChua1 khi ở chế độ Sim Mode
   RUNG wire#powerrail
      Contact( "HMI_Sim_Mode" )
      Contact( "TT3301_BonChua1_Sim_Req" )
      Coil( "TT3301_BonChua1_Sim_Active" )
   END_RUNG
   // the same network as SCL:
   "TT3301_BonChua1_Sim_Active" := "HMI_Sim_Mode" AND "TT3301_BonChua1_Sim_Req";
END_REGION

REGION Network 11: Đọc giá trị mô phỏng TT3301_BonChua1 vào hiệu dụng
   RUNG wire#powerrail
      Contact( "TT3301_BonChua1_Sim_Active" )
      { S7_GenerateENO := "TRUE" } Move(in := "TT3301_BonChua1_HMI", out1 => "TT3301_BonChua1_Eff")
   END_RUNG
   // the same network as SCL:
   IF "TT3301_BonChua1_Sim_Active" THEN "TT3301_BonChua1_Eff" := "TT3301_BonChua1_HMI"; END_IF;
END_REGION

REGION Network 12: Đọc giá trị vật lý TT3301_BonChua1 vào hiệu dụng
   RUNG wire#powerrail
      I_Contact( "TT3301_BonChua1_Sim_Active" )
      { S7_GenerateENO := "TRUE" } Move(in := "TT3301_BonChua1", out1 => "TT3301_BonChua1_Eff")
   END_RUNG
   // the same network as SCL:
   IF NOT "TT3301_BonChua1_Sim_Active" THEN "TT3301_BonChua1_Eff" := "TT3301_BonChua1"; END_IF;
END_REGION

REGION Network 13: Yêu cầu mô phỏng TT3303_TraoDoiNhiet từ HMI
   RUNG wire#powerrail
      Contact( "HMI_Use_Sim_Input_BonChua" )
      wire#w1
      Coil( "TT3303_TraoDoiNhiet_Sim_Req" )
   END_RUNG
   RUNG wire#powerrail
      Contact( "TT3303_TraoDoiNhiet_Use_HMI" )
   END_RUNG wire#w1
   // the same network as SCL:
   "TT3303_TraoDoiNhiet_Sim_Req" := "HMI_Use_Sim_Input_BonChua" OR "TT3303_TraoDoiNhiet_Use_HMI";
END_REGION

REGION Network 14: Kích hoạt mô phỏng TT3303_TraoDoiNhiet khi ở chế độ Sim Mode
   RUNG wire#powerrail
      Contact( "HMI_Sim_Mode" )
      Contact( "TT3303_TraoDoiNhiet_Sim_Req" )
      Coil( "TT3303_TraoDoiNhiet_Sim_Active" )
   END_RUNG
   // the same network as SCL:
   "TT3303_TraoDoiNhiet_Sim_Active" := "HMI_Sim_Mode" AND "TT3303_TraoDoiNhiet_Sim_Req";
END_REGION

REGION Network 15: Đọc giá trị mô phỏng TT3303_TraoDoiNhiet vào hiệu dụng
   RUNG wire#powerrail
      Contact( "TT3303_TraoDoiNhiet_Sim_Active" )
      { S7_GenerateENO := "TRUE" } Move(in := "TT3303_TraoDoiNhiet_HMI", out1 => "TT3303_TraoDoiNhiet_Eff")
   END_RUNG
   // the same network as SCL:
   IF "TT3303_TraoDoiNhiet_Sim_Active" THEN "TT3303_TraoDoiNhiet_Eff" := "TT3303_TraoDoiNhiet_HMI"; END_IF;
END_REGION

REGION Network 16: Đọc giá trị vật lý TT3303_TraoDoiNhiet vào hiệu dụng
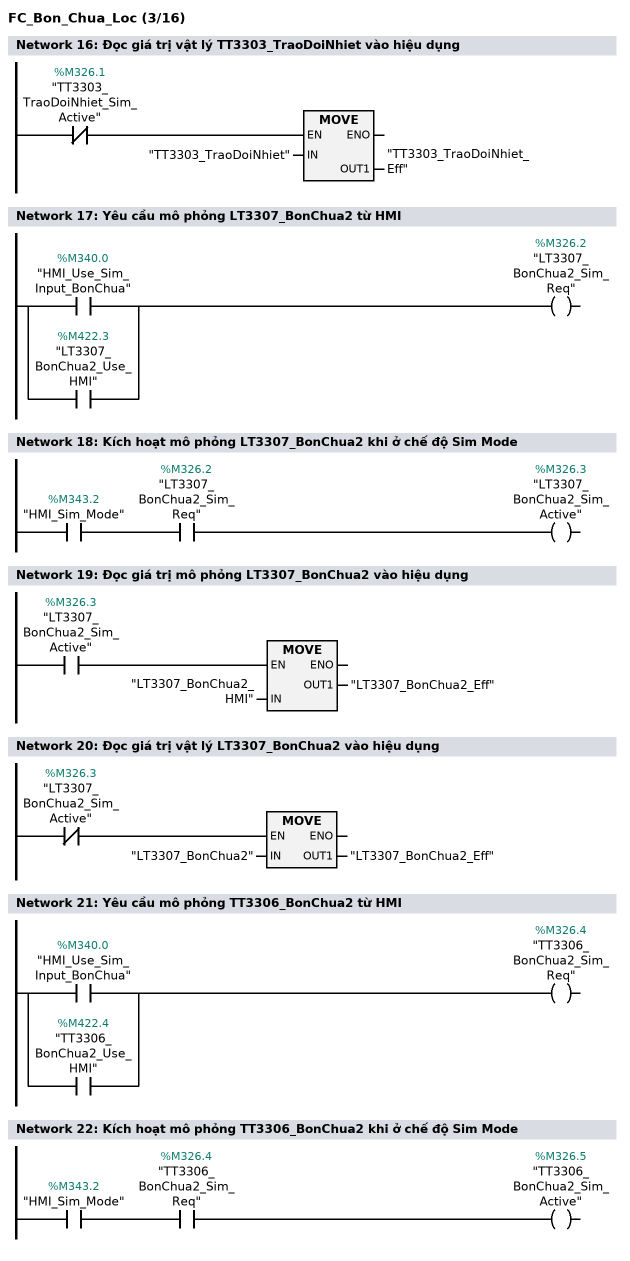
   RUNG wire#powerrail
      I_Contact( "TT3303_TraoDoiNhiet_Sim_Active" )
      { S7_GenerateENO := "TRUE" } Move(in := "TT3303_TraoDoiNhiet", out1 => "TT3303_TraoDoiNhiet_Eff")
   END_RUNG
   // the same network as SCL:
   IF NOT "TT3303_TraoDoiNhiet_Sim_Active" THEN "TT3303_TraoDoiNhiet_Eff" := "TT3303_TraoDoiNhiet"; END_IF;
END_REGION

REGION Network 17: Yêu cầu mô phỏng LT3307_BonChua2 từ HMI
   RUNG wire#powerrail
      Contact( "HMI_Use_Sim_Input_BonChua" )
      wire#w1
      Coil( "LT3307_BonChua2_Sim_Req" )
   END_RUNG
   RUNG wire#powerrail
      Contact( "LT3307_BonChua2_Use_HMI" )
   END_RUNG wire#w1
   // the same network as SCL:
   "LT3307_BonChua2_Sim_Req" := "HMI_Use_Sim_Input_BonChua" OR "LT3307_BonChua2_Use_HMI";
END_REGION

REGION Network 18: Kích hoạt mô phỏng LT3307_BonChua2 khi ở chế độ Sim Mode
   RUNG wire#powerrail
      Contact( "HMI_Sim_Mode" )
      Contact( "LT3307_BonChua2_Sim_Req" )
      Coil( "LT3307_BonChua2_Sim_Active" )
   END_RUNG
   // the same network as SCL:
   "LT3307_BonChua2_Sim_Active" := "HMI_Sim_Mode" AND "LT3307_BonChua2_Sim_Req";
END_REGION

REGION Network 19: Đọc giá trị mô phỏng LT3307_BonChua2 vào hiệu dụng
   RUNG wire#powerrail
      Contact( "LT3307_BonChua2_Sim_Active" )
      { S7_GenerateENO := "TRUE" } Move(in := "LT3307_BonChua2_HMI", out1 => "LT3307_BonChua2_Eff")
   END_RUNG
   // the same network as SCL:
   IF "LT3307_BonChua2_Sim_Active" THEN "LT3307_BonChua2_Eff" := "LT3307_BonChua2_HMI"; END_IF;
END_REGION

REGION Network 20: Đọc giá trị vật lý LT3307_BonChua2 vào hiệu dụng
   RUNG wire#powerrail
      I_Contact( "LT3307_BonChua2_Sim_Active" )
      { S7_GenerateENO := "TRUE" } Move(in := "LT3307_BonChua2", out1 => "LT3307_BonChua2_Eff")
   END_RUNG
   // the same network as SCL:
   IF NOT "LT3307_BonChua2_Sim_Active" THEN "LT3307_BonChua2_Eff" := "LT3307_BonChua2"; END_IF;
END_REGION

REGION Network 21: Yêu cầu mô phỏng TT3306_BonChua2 từ HMI
   RUNG wire#powerrail
      Contact( "HMI_Use_Sim_Input_BonChua" )
      wire#w1
      Coil( "TT3306_BonChua2_Sim_Req" )
   END_RUNG
   RUNG wire#powerrail
      Contact( "TT3306_BonChua2_Use_HMI" )
   END_RUNG wire#w1
   // the same network as SCL:
   "TT3306_BonChua2_Sim_Req" := "HMI_Use_Sim_Input_BonChua" OR "TT3306_BonChua2_Use_HMI";
END_REGION

REGION Network 22: Kích hoạt mô phỏng TT3306_BonChua2 khi ở chế độ Sim Mode
   RUNG wire#powerrail
      Contact( "HMI_Sim_Mode" )
      Contact( "TT3306_BonChua2_Sim_Req" )
      Coil( "TT3306_BonChua2_Sim_Active" )
   END_RUNG
   // the same network as SCL:
   "TT3306_BonChua2_Sim_Active" := "HMI_Sim_Mode" AND "TT3306_BonChua2_Sim_Req";
END_REGION

REGION Network 23: Đọc giá trị mô phỏng TT3306_BonChua2 vào hiệu dụng
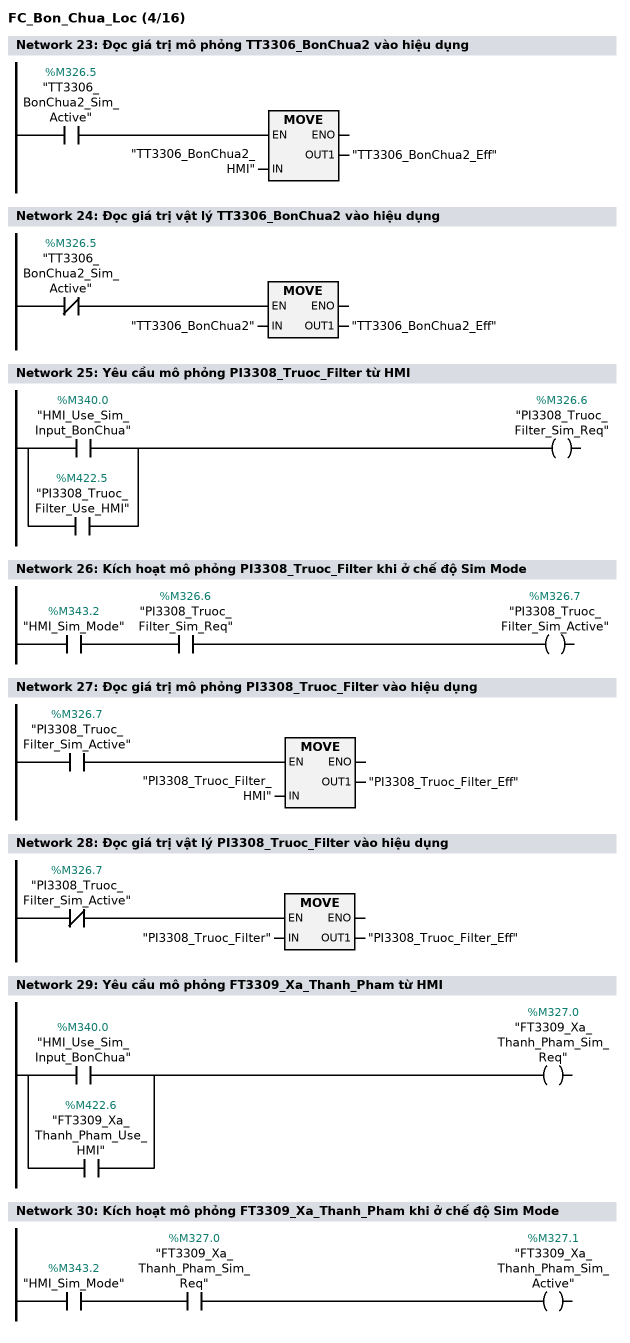
   RUNG wire#powerrail
      Contact( "TT3306_BonChua2_Sim_Active" )
      { S7_GenerateENO := "TRUE" } Move(in := "TT3306_BonChua2_HMI", out1 => "TT3306_BonChua2_Eff")
   END_RUNG
   // the same network as SCL:
   IF "TT3306_BonChua2_Sim_Active" THEN "TT3306_BonChua2_Eff" := "TT3306_BonChua2_HMI"; END_IF;
END_REGION

REGION Network 24: Đọc giá trị vật lý TT3306_BonChua2 vào hiệu dụng
   RUNG wire#powerrail
      I_Contact( "TT3306_BonChua2_Sim_Active" )
      { S7_GenerateENO := "TRUE" } Move(in := "TT3306_BonChua2", out1 => "TT3306_BonChua2_Eff")
   END_RUNG
   // the same network as SCL:
   IF NOT "TT3306_BonChua2_Sim_Active" THEN "TT3306_BonChua2_Eff" := "TT3306_BonChua2"; END_IF;
END_REGION

REGION Network 25: Yêu cầu mô phỏng PI3308_Truoc_Filter từ HMI
   RUNG wire#powerrail
      Contact( "HMI_Use_Sim_Input_BonChua" )
      wire#w1
      Coil( "PI3308_Truoc_Filter_Sim_Req" )
   END_RUNG
   RUNG wire#powerrail
      Contact( "PI3308_Truoc_Filter_Use_HMI" )
   END_RUNG wire#w1
   // the same network as SCL:
   "PI3308_Truoc_Filter_Sim_Req" := "HMI_Use_Sim_Input_BonChua" OR "PI3308_Truoc_Filter_Use_HMI";
END_REGION

REGION Network 26: Kích hoạt mô phỏng PI3308_Truoc_Filter khi ở chế độ Sim Mode
   RUNG wire#powerrail
      Contact( "HMI_Sim_Mode" )
      Contact( "PI3308_Truoc_Filter_Sim_Req" )
      Coil( "PI3308_Truoc_Filter_Sim_Active" )
   END_RUNG
   // the same network as SCL:
   "PI3308_Truoc_Filter_Sim_Active" := "HMI_Sim_Mode" AND "PI3308_Truoc_Filter_Sim_Req";
END_REGION

REGION Network 27: Đọc giá trị mô phỏng PI3308_Truoc_Filter vào hiệu dụng
   RUNG wire#powerrail
      Contact( "PI3308_Truoc_Filter_Sim_Active" )
      { S7_GenerateENO := "TRUE" } Move(in := "PI3308_Truoc_Filter_HMI", out1 => "PI3308_Truoc_Filter_Eff")
   END_RUNG
   // the same network as SCL:
   IF "PI3308_Truoc_Filter_Sim_Active" THEN "PI3308_Truoc_Filter_Eff" := "PI3308_Truoc_Filter_HMI"; END_IF;
END_REGION

REGION Network 28: Đọc giá trị vật lý PI3308_Truoc_Filter vào hiệu dụng
   RUNG wire#powerrail
      I_Contact( "PI3308_Truoc_Filter_Sim_Active" )
      { S7_GenerateENO := "TRUE" } Move(in := "PI3308_Truoc_Filter", out1 => "PI3308_Truoc_Filter_Eff")
   END_RUNG
   // the same network as SCL:
   IF NOT "PI3308_Truoc_Filter_Sim_Active" THEN "PI3308_Truoc_Filter_Eff" := "PI3308_Truoc_Filter"; END_IF;
END_REGION

REGION Network 29: Yêu cầu mô phỏng FT3309_Xa_Thanh_Pham từ HMI
   RUNG wire#powerrail
      Contact( "HMI_Use_Sim_Input_BonChua" )
      wire#w1
      Coil( "FT3309_Xa_Thanh_Pham_Sim_Req" )
   END_RUNG
   RUNG wire#powerrail
      Contact( "FT3309_Xa_Thanh_Pham_Use_HMI" )
   END_RUNG wire#w1
   // the same network as SCL:
   "FT3309_Xa_Thanh_Pham_Sim_Req" := "HMI_Use_Sim_Input_BonChua" OR "FT3309_Xa_Thanh_Pham_Use_HMI";
END_REGION

REGION Network 30: Kích hoạt mô phỏng FT3309_Xa_Thanh_Pham khi ở chế độ Sim Mode
   RUNG wire#powerrail
      Contact( "HMI_Sim_Mode" )
      Contact( "FT3309_Xa_Thanh_Pham_Sim_Req" )
      Coil( "FT3309_Xa_Thanh_Pham_Sim_Active" )
   END_RUNG
   // the same network as SCL:
   "FT3309_Xa_Thanh_Pham_Sim_Active" := "HMI_Sim_Mode" AND "FT3309_Xa_Thanh_Pham_Sim_Req";
END_REGION

REGION Network 31: Đọc giá trị mô phỏng FT3309_Xa_Thanh_Pham vào hiệu dụng
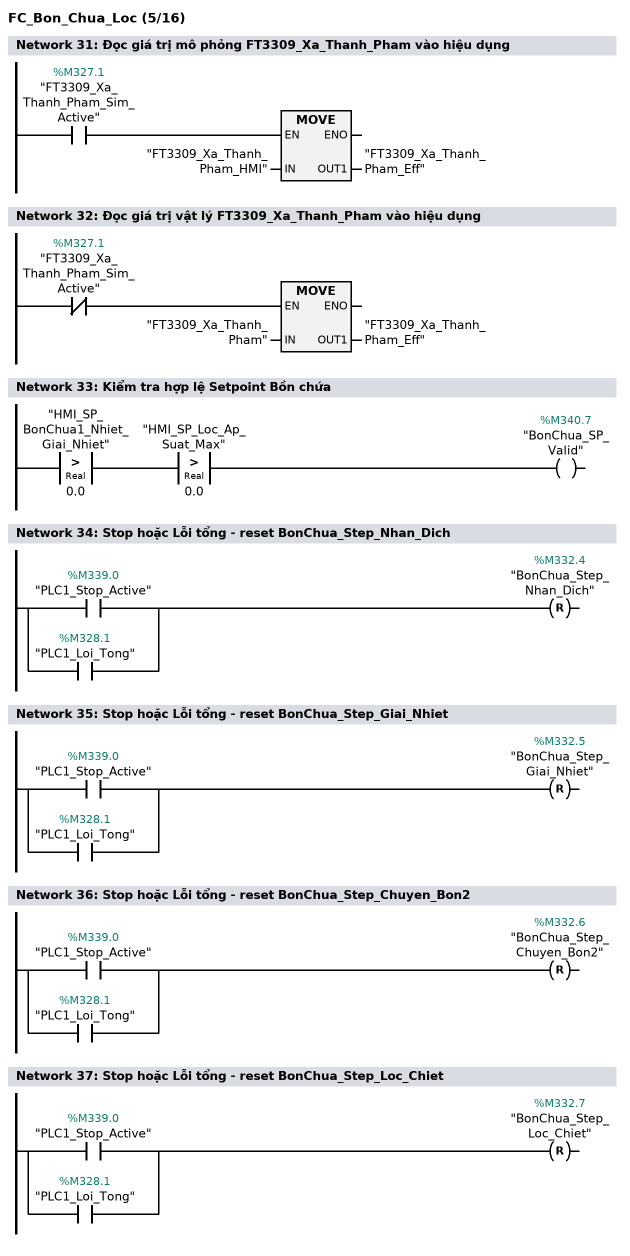
   RUNG wire#powerrail
      Contact( "FT3309_Xa_Thanh_Pham_Sim_Active" )
      { S7_GenerateENO := "TRUE" } Move(in := "FT3309_Xa_Thanh_Pham_HMI", out1 => "FT3309_Xa_Thanh_Pham_Eff")
   END_RUNG
   // the same network as SCL:
   IF "FT3309_Xa_Thanh_Pham_Sim_Active" THEN
       "FT3309_Xa_Thanh_Pham_Eff" := "FT3309_Xa_Thanh_Pham_HMI";
   END_IF;
END_REGION

REGION Network 32: Đọc giá trị vật lý FT3309_Xa_Thanh_Pham vào hiệu dụng
   RUNG wire#powerrail
      I_Contact( "FT3309_Xa_Thanh_Pham_Sim_Active" )
      { S7_GenerateENO := "TRUE" } Move(in := "FT3309_Xa_Thanh_Pham", out1 => "FT3309_Xa_Thanh_Pham_Eff")
   END_RUNG
   // the same network as SCL:
   IF NOT "FT3309_Xa_Thanh_Pham_Sim_Active" THEN
       "FT3309_Xa_Thanh_Pham_Eff" := "FT3309_Xa_Thanh_Pham";
   END_IF;
END_REGION

REGION Network 33: Kiểm tra hợp lệ Setpoint Bồn chứa
   RUNG wire#powerrail
      { S7_Templates := "SrcType := Real" } GT_Contact(in1 := "HMI_SP_BonChua1_Nhiet_Giai_Nhiet", in2 := 0.0)
      { S7_Templates := "SrcType := Real" } GT_Contact(in1 := "HMI_SP_Loc_Ap_Suat_Max", in2 := 0.0)
      Coil( "BonChua_SP_Valid" )
   END_RUNG
   // the same network as SCL:
   "BonChua_SP_Valid" := ("HMI_SP_BonChua1_Nhiet_Giai_Nhiet" > 0.0) AND ("HMI_SP_Loc_Ap_Suat_Max" > 0.0);
END_REGION

REGION Network 34: Stop hoặc Lỗi tổng - reset BonChua_Step_Nhan_Dich
   RUNG wire#powerrail
      Contact( "PLC1_Stop_Active" )
      wire#w1
      R_Coil( "BonChua_Step_Nhan_Dich" )
   END_RUNG
   RUNG wire#powerrail
      Contact( "PLC1_Loi_Tong" )
   END_RUNG wire#w1
   // the same network as SCL:
   IF "PLC1_Stop_Active" OR "PLC1_Loi_Tong" THEN "BonChua_Step_Nhan_Dich" := FALSE; END_IF;
END_REGION

REGION Network 35: Stop hoặc Lỗi tổng - reset BonChua_Step_Giai_Nhiet
   RUNG wire#powerrail
      Contact( "PLC1_Stop_Active" )
      wire#w1
      R_Coil( "BonChua_Step_Giai_Nhiet" )
   END_RUNG
   RUNG wire#powerrail
      Contact( "PLC1_Loi_Tong" )
   END_RUNG wire#w1
   // the same network as SCL:
   IF "PLC1_Stop_Active" OR "PLC1_Loi_Tong" THEN "BonChua_Step_Giai_Nhiet" := FALSE; END_IF;
END_REGION

REGION Network 36: Stop hoặc Lỗi tổng - reset BonChua_Step_Chuyen_Bon2
   RUNG wire#powerrail
      Contact( "PLC1_Stop_Active" )
      wire#w1
      R_Coil( "BonChua_Step_Chuyen_Bon2" )
   END_RUNG
   RUNG wire#powerrail
      Contact( "PLC1_Loi_Tong" )
   END_RUNG wire#w1
   // the same network as SCL:
   IF "PLC1_Stop_Active" OR "PLC1_Loi_Tong" THEN "BonChua_Step_Chuyen_Bon2" := FALSE; END_IF;
END_REGION

REGION Network 37: Stop hoặc Lỗi tổng - reset BonChua_Step_Loc_Chiet
   RUNG wire#powerrail
      Contact( "PLC1_Stop_Active" )
      wire#w1
      R_Coil( "BonChua_Step_Loc_Chiet" )
   END_RUNG
   RUNG wire#powerrail
      Contact( "PLC1_Loi_Tong" )
   END_RUNG wire#w1
   // the same network as SCL:
   IF "PLC1_Stop_Active" OR "PLC1_Loi_Tong" THEN "BonChua_Step_Loc_Chiet" := FALSE; END_IF;
END_REGION

REGION Network 38: Stop hoặc Lỗi tổng - reset BonChua_Me_Hoan_Thanh
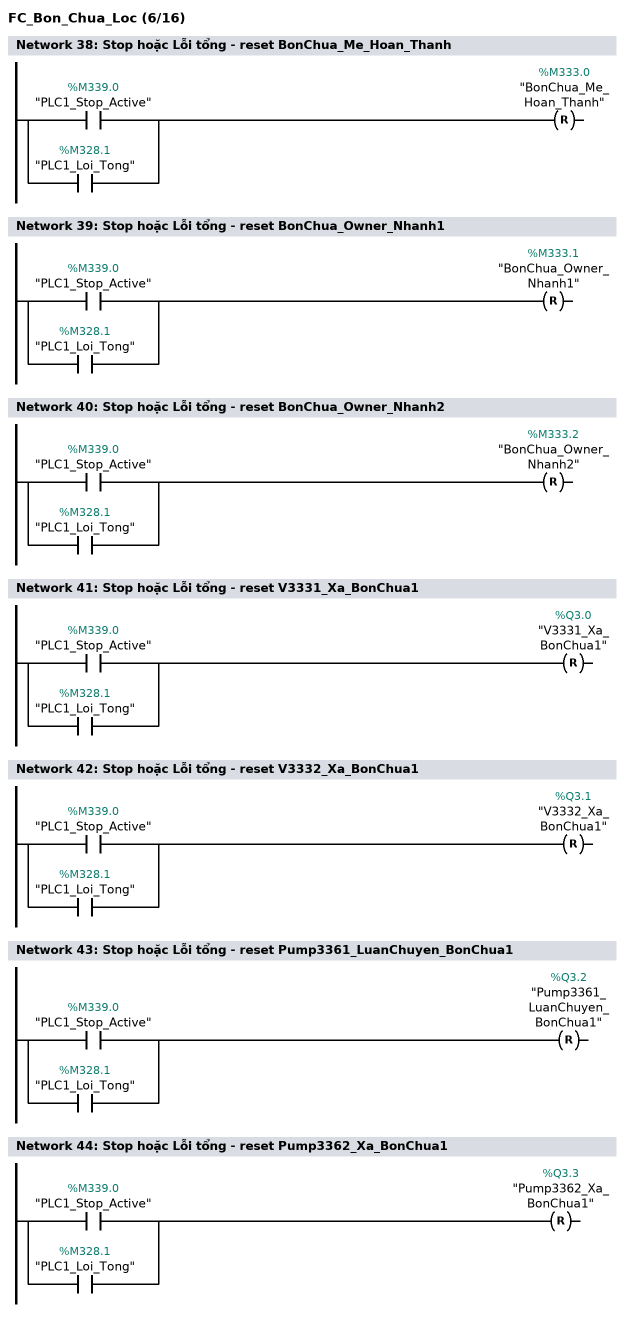
   RUNG wire#powerrail
      Contact( "PLC1_Stop_Active" )
      wire#w1
      R_Coil( "BonChua_Me_Hoan_Thanh" )
   END_RUNG
   RUNG wire#powerrail
      Contact( "PLC1_Loi_Tong" )
   END_RUNG wire#w1
   // the same network as SCL:
   IF "PLC1_Stop_Active" OR "PLC1_Loi_Tong" THEN "BonChua_Me_Hoan_Thanh" := FALSE; END_IF;
END_REGION

REGION Network 39: Stop hoặc Lỗi tổng - reset BonChua_Owner_Nhanh1
   RUNG wire#powerrail
      Contact( "PLC1_Stop_Active" )
      wire#w1
      R_Coil( "BonChua_Owner_Nhanh1" )
   END_RUNG
   RUNG wire#powerrail
      Contact( "PLC1_Loi_Tong" )
   END_RUNG wire#w1
   // the same network as SCL:
   IF "PLC1_Stop_Active" OR "PLC1_Loi_Tong" THEN "BonChua_Owner_Nhanh1" := FALSE; END_IF;
END_REGION

REGION Network 40: Stop hoặc Lỗi tổng - reset BonChua_Owner_Nhanh2
   RUNG wire#powerrail
      Contact( "PLC1_Stop_Active" )
      wire#w1
      R_Coil( "BonChua_Owner_Nhanh2" )
   END_RUNG
   RUNG wire#powerrail
      Contact( "PLC1_Loi_Tong" )
   END_RUNG wire#w1
   // the same network as SCL:
   IF "PLC1_Stop_Active" OR "PLC1_Loi_Tong" THEN "BonChua_Owner_Nhanh2" := FALSE; END_IF;
END_REGION

REGION Network 41: Stop hoặc Lỗi tổng - reset V3331_Xa_BonChua1
   RUNG wire#powerrail
      Contact( "PLC1_Stop_Active" )
      wire#w1
      R_Coil( "V3331_Xa_BonChua1" )
   END_RUNG
   RUNG wire#powerrail
      Contact( "PLC1_Loi_Tong" )
   END_RUNG wire#w1
   // the same network as SCL:
   IF "PLC1_Stop_Active" OR "PLC1_Loi_Tong" THEN "V3331_Xa_BonChua1" := FALSE; END_IF;
END_REGION

REGION Network 42: Stop hoặc Lỗi tổng - reset V3332_Xa_BonChua1
   RUNG wire#powerrail
      Contact( "PLC1_Stop_Active" )
      wire#w1
      R_Coil( "V3332_Xa_BonChua1" )
   END_RUNG
   RUNG wire#powerrail
      Contact( "PLC1_Loi_Tong" )
   END_RUNG wire#w1
   // the same network as SCL:
   IF "PLC1_Stop_Active" OR "PLC1_Loi_Tong" THEN "V3332_Xa_BonChua1" := FALSE; END_IF;
END_REGION

REGION Network 43: Stop hoặc Lỗi tổng - reset Pump3361_LuanChuyen_BonChua1
   RUNG wire#powerrail
      Contact( "PLC1_Stop_Active" )
      wire#w1
      R_Coil( "Pump3361_LuanChuyen_BonChua1" )
   END_RUNG
   RUNG wire#powerrail
      Contact( "PLC1_Loi_Tong" )
   END_RUNG wire#w1
   // the same network as SCL:
   IF "PLC1_Stop_Active" OR "PLC1_Loi_Tong" THEN "Pump3361_LuanChuyen_BonChua1" := FALSE; END_IF;
END_REGION

REGION Network 44: Stop hoặc Lỗi tổng - reset Pump3362_Xa_BonChua1
   RUNG wire#powerrail
      Contact( "PLC1_Stop_Active" )
      wire#w1
      R_Coil( "Pump3362_Xa_BonChua1" )
   END_RUNG
   RUNG wire#powerrail
      Contact( "PLC1_Loi_Tong" )
   END_RUNG wire#w1
   // the same network as SCL:
   IF "PLC1_Stop_Active" OR "PLC1_Loi_Tong" THEN "Pump3362_Xa_BonChua1" := FALSE; END_IF;
END_REGION

REGION Network 45: Stop hoặc Lỗi tổng - reset V3333_DieuHuong_BonChua1
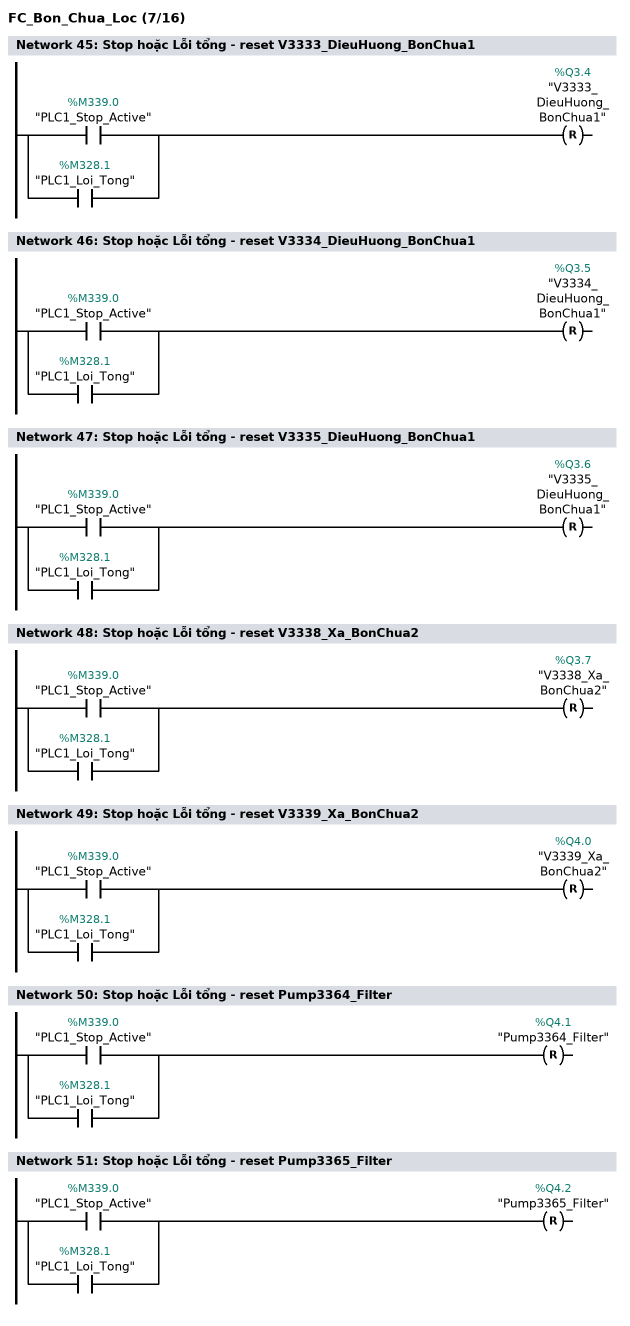
   RUNG wire#powerrail
      Contact( "PLC1_Stop_Active" )
      wire#w1
      R_Coil( "V3333_DieuHuong_BonChua1" )
   END_RUNG
   RUNG wire#powerrail
      Contact( "PLC1_Loi_Tong" )
   END_RUNG wire#w1
   // the same network as SCL:
   IF "PLC1_Stop_Active" OR "PLC1_Loi_Tong" THEN "V3333_DieuHuong_BonChua1" := FALSE; END_IF;
END_REGION

REGION Network 46: Stop hoặc Lỗi tổng - reset V3334_DieuHuong_BonChua1
   RUNG wire#powerrail
      Contact( "PLC1_Stop_Active" )
      wire#w1
      R_Coil( "V3334_DieuHuong_BonChua1" )
   END_RUNG
   RUNG wire#powerrail
      Contact( "PLC1_Loi_Tong" )
   END_RUNG wire#w1
   // the same network as SCL:
   IF "PLC1_Stop_Active" OR "PLC1_Loi_Tong" THEN "V3334_DieuHuong_BonChua1" := FALSE; END_IF;
END_REGION

REGION Network 47: Stop hoặc Lỗi tổng - reset V3335_DieuHuong_BonChua1
   RUNG wire#powerrail
      Contact( "PLC1_Stop_Active" )
      wire#w1
      R_Coil( "V3335_DieuHuong_BonChua1" )
   END_RUNG
   RUNG wire#powerrail
      Contact( "PLC1_Loi_Tong" )
   END_RUNG wire#w1
   // the same network as SCL:
   IF "PLC1_Stop_Active" OR "PLC1_Loi_Tong" THEN "V3335_DieuHuong_BonChua1" := FALSE; END_IF;
END_REGION

REGION Network 48: Stop hoặc Lỗi tổng - reset V3338_Xa_BonChua2
   RUNG wire#powerrail
      Contact( "PLC1_Stop_Active" )
      wire#w1
      R_Coil( "V3338_Xa_BonChua2" )
   END_RUNG
   RUNG wire#powerrail
      Contact( "PLC1_Loi_Tong" )
   END_RUNG wire#w1
   // the same network as SCL:
   IF "PLC1_Stop_Active" OR "PLC1_Loi_Tong" THEN "V3338_Xa_BonChua2" := FALSE; END_IF;
END_REGION

REGION Network 49: Stop hoặc Lỗi tổng - reset V3339_Xa_BonChua2
   RUNG wire#powerrail
      Contact( "PLC1_Stop_Active" )
      wire#w1
      R_Coil( "V3339_Xa_BonChua2" )
   END_RUNG
   RUNG wire#powerrail
      Contact( "PLC1_Loi_Tong" )
   END_RUNG wire#w1
   // the same network as SCL:
   IF "PLC1_Stop_Active" OR "PLC1_Loi_Tong" THEN "V3339_Xa_BonChua2" := FALSE; END_IF;
END_REGION

REGION Network 50: Stop hoặc Lỗi tổng - reset Pump3364_Filter
   RUNG wire#powerrail
      Contact( "PLC1_Stop_Active" )
      wire#w1
      R_Coil( "Pump3364_Filter" )
   END_RUNG
   RUNG wire#powerrail
      Contact( "PLC1_Loi_Tong" )
   END_RUNG wire#w1
   // the same network as SCL:
   IF "PLC1_Stop_Active" OR "PLC1_Loi_Tong" THEN "Pump3364_Filter" := FALSE; END_IF;
END_REGION

REGION Network 51: Stop hoặc Lỗi tổng - reset Pump3365_Filter
   RUNG wire#powerrail
      Contact( "PLC1_Stop_Active" )
      wire#w1
      R_Coil( "Pump3365_Filter" )
   END_RUNG
   RUNG wire#powerrail
      Contact( "PLC1_Loi_Tong" )
   END_RUNG wire#w1
   // the same network as SCL:
   IF "PLC1_Stop_Active" OR "PLC1_Loi_Tong" THEN "Pump3365_Filter" := FALSE; END_IF;
END_REGION

REGION Network 52: Stop hoặc Lỗi tổng - reset V3340_Duong_Filter
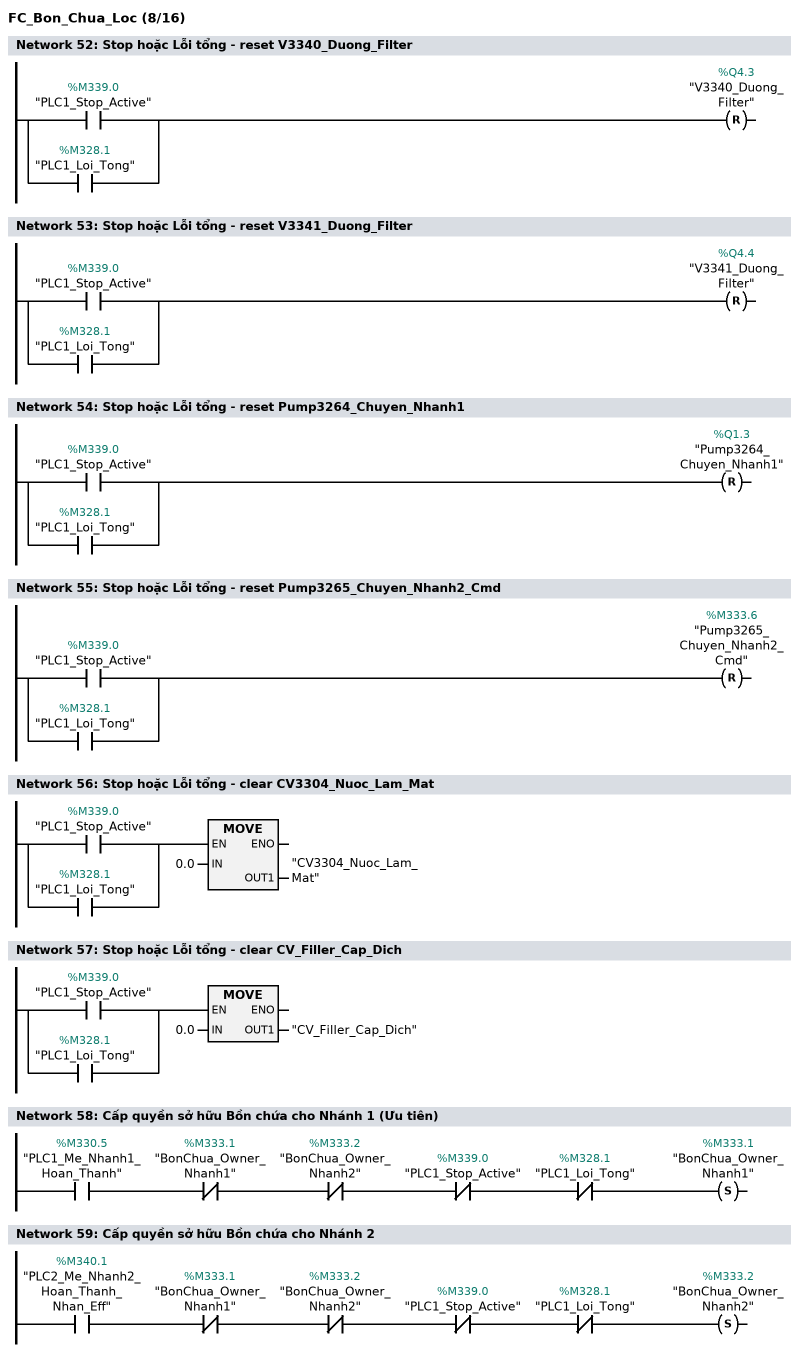
   RUNG wire#powerrail
      Contact( "PLC1_Stop_Active" )
      wire#w1
      R_Coil( "V3340_Duong_Filter" )
   END_RUNG
   RUNG wire#powerrail
      Contact( "PLC1_Loi_Tong" )
   END_RUNG wire#w1
   // the same network as SCL:
   IF "PLC1_Stop_Active" OR "PLC1_Loi_Tong" THEN "V3340_Duong_Filter" := FALSE; END_IF;
END_REGION

REGION Network 53: Stop hoặc Lỗi tổng - reset V3341_Duong_Filter
   RUNG wire#powerrail
      Contact( "PLC1_Stop_Active" )
      wire#w1
      R_Coil( "V3341_Duong_Filter" )
   END_RUNG
   RUNG wire#powerrail
      Contact( "PLC1_Loi_Tong" )
   END_RUNG wire#w1
   // the same network as SCL:
   IF "PLC1_Stop_Active" OR "PLC1_Loi_Tong" THEN "V3341_Duong_Filter" := FALSE; END_IF;
END_REGION

REGION Network 54: Stop hoặc Lỗi tổng - reset Pump3264_Chuyen_Nhanh1
   RUNG wire#powerrail
      Contact( "PLC1_Stop_Active" )
      wire#w1
      R_Coil( "Pump3264_Chuyen_Nhanh1" )
   END_RUNG
   RUNG wire#powerrail
      Contact( "PLC1_Loi_Tong" )
   END_RUNG wire#w1
   // the same network as SCL:
   IF "PLC1_Stop_Active" OR "PLC1_Loi_Tong" THEN "Pump3264_Chuyen_Nhanh1" := FALSE; END_IF;
END_REGION

REGION Network 55: Stop hoặc Lỗi tổng - reset Pump3265_Chuyen_Nhanh2_Cmd
   RUNG wire#powerrail
      Contact( "PLC1_Stop_Active" )
      wire#w1
      R_Coil( "Pump3265_Chuyen_Nhanh2_Cmd" )
   END_RUNG
   RUNG wire#powerrail
      Contact( "PLC1_Loi_Tong" )
   END_RUNG wire#w1
   // the same network as SCL:
   IF "PLC1_Stop_Active" OR "PLC1_Loi_Tong" THEN "Pump3265_Chuyen_Nhanh2_Cmd" := FALSE; END_IF;
END_REGION

REGION Network 56: Stop hoặc Lỗi tổng - clear CV3304_Nuoc_Lam_Mat
   RUNG wire#powerrail
      Contact( "PLC1_Stop_Active" )
      wire#w1
      { S7_GenerateENO := "TRUE" } Move(in := 0.0, out1 => "CV3304_Nuoc_Lam_Mat")
   END_RUNG
   RUNG wire#powerrail
      Contact( "PLC1_Loi_Tong" )
   END_RUNG wire#w1
   // the same network as SCL:
   IF "PLC1_Stop_Active" OR "PLC1_Loi_Tong" THEN "CV3304_Nuoc_Lam_Mat" := 0.0; END_IF;
END_REGION

REGION Network 57: Stop hoặc Lỗi tổng - clear CV_Filler_Cap_Dich
   RUNG wire#powerrail
      Contact( "PLC1_Stop_Active" )
      wire#w1
      { S7_GenerateENO := "TRUE" } Move(in := 0.0, out1 => "CV_Filler_Cap_Dich")
   END_RUNG
   RUNG wire#powerrail
      Contact( "PLC1_Loi_Tong" )
   END_RUNG wire#w1
   // the same network as SCL:
   IF "PLC1_Stop_Active" OR "PLC1_Loi_Tong" THEN "CV_Filler_Cap_Dich" := 0.0; END_IF;
END_REGION

REGION Network 58: Cấp quyền sở hữu Bồn chứa cho Nhánh 1 (Ưu tiên)
   RUNG wire#powerrail
      Contact( "PLC1_Me_Nhanh1_Hoan_Thanh" )
      I_Contact( "BonChua_Owner_Nhanh1" )
      I_Contact( "BonChua_Owner_Nhanh2" )
      I_Contact( "PLC1_Stop_Active" )
      I_Contact( "PLC1_Loi_Tong" )
      S_Coil( "BonChua_Owner_Nhanh1" )
   END_RUNG
   // the same network as SCL:
   IF "PLC1_Me_Nhanh1_Hoan_Thanh" AND NOT "BonChua_Owner_Nhanh1" AND NOT "BonChua_Owner_Nhanh2" AND NOT "PLC1_Stop_Active" AND NOT "PLC1_Loi_Tong" THEN
       "BonChua_Owner_Nhanh1" := TRUE;
   END_IF;
END_REGION

REGION Network 59: Cấp quyền sở hữu Bồn chứa cho Nhánh 2
   RUNG wire#powerrail
      Contact( "PLC2_Me_Nhanh2_Hoan_Thanh_Nhan_Eff" )
      I_Contact( "BonChua_Owner_Nhanh1" )
      I_Contact( "BonChua_Owner_Nhanh2" )
      I_Contact( "PLC1_Stop_Active" )
      I_Contact( "PLC1_Loi_Tong" )
      S_Coil( "BonChua_Owner_Nhanh2" )
   END_RUNG
   // the same network as SCL:
   IF "PLC2_Me_Nhanh2_Hoan_Thanh_Nhan_Eff" AND NOT "BonChua_Owner_Nhanh1" AND NOT "BonChua_Owner_Nhanh2" AND NOT "PLC1_Stop_Active" AND NOT "PLC1_Loi_Tong" THEN
       "BonChua_Owner_Nhanh2" := TRUE;
   END_IF;
END_REGION

REGION Network 60: Bản đồ trạng thái Storage - Nhận dịch (State 50)
